// TIA Portal V20 program export: 0 tag tables, 0 data types, 5 data blocks, 15 code blocks (in call order from the OBs), 9 instance data blocks

DATA_BLOCK "Data_State2"   // DB12
{ S7_Optimized_Access := 'FALSE' }
   VAR
      state1 : "UDT_Flowmeter_Status";
      state_2 : "UDT_Flowmeter_Stoe";
   END_VAR
BEGIN
END_DATA_BLOCK

DATA_BLOCK "Date and Time"   // DB3
{ S7_Optimized_Access := 'FALSE' }
AUTHOR : L.P.
// stored: AutoNumber false
   VAR RETAIN
      MEM : Struct
         "set by host" : Bool;
         "HM imp set by host" : Bool;
         "HM imp set by HMI" : Bool := false;
         "4" : Bool := false;
         "5" : Bool := false;
         "6" : Bool := false;
         "7" : Bool := false;
         "8" : Bool := false;
         "9" : Bool := false;
         "10" : Bool := false;
      END_STRUCT;
      "STEP" : Struct
         "0" : Bool;
         "1" : Bool;
         "2" : Bool;
         "3" : Bool;
         "4" : Bool;
         "5" : Bool;
         "6" : Bool;
         "7" : Bool;
         "8" : Bool;
         "9" : Bool;
         "10" : Bool;
      END_STRUCT;
      T : Struct
         "1" { S7_SetPoint := 'True'} : IEC_TIMER;
         "2" { S7_SetPoint := 'True'} : IEC_TIMER;
         "3" { S7_SetPoint := 'True'} : IEC_TIMER;
         "4" { S7_SetPoint := 'True'} : IEC_TIMER;
         "5" { S7_SetPoint := 'True'} : IEC_TIMER;
         "6" { S7_SetPoint := 'True'} : IEC_TIMER;
         "7" { S7_SetPoint := 'True'} : IEC_TIMER;
         "8" { S7_SetPoint := 'True'} : IEC_TIMER;
         "9" { S7_SetPoint := 'True'} : IEC_TIMER;
         "10" { S7_SetPoint := 'True'} : IEC_TIMER;
      END_STRUCT;
      C : Struct
         "1" { S7_SetPoint := 'True'} : IEC_COUNTER;
         "2" { S7_SetPoint := 'True'} : IEC_COUNTER;
         "3" { S7_SetPoint := 'True'} : IEC_COUNTER;
         "4" { S7_SetPoint := 'True'} : IEC_COUNTER;
         "5" { S7_SetPoint := 'True'} : IEC_COUNTER;
         "6" { S7_SetPoint := 'True'} : IEC_COUNTER;
         "7" { S7_SetPoint := 'True'} : IEC_COUNTER;
         "8" { S7_SetPoint := 'True'} : IEC_COUNTER;
         "9" { S7_SetPoint := 'True'} : IEC_COUNTER;
         "10" { S7_SetPoint := 'True'} : IEC_COUNTER;
      END_STRUCT;
      DATA : Struct
         "in date OP" : Date;
         "in time OP" : Time_Of_Day;
         "in date and time" : DTL;
         "out date and time" : DTL;
         year : UInt;
         month : USInt;
         day : USInt;
         hour : USInt;
         minute : USInt;
         second : USInt;
         millisecond : UInt;
         "day of week" : USInt;
         "day of year" : Int;
         "is Time Master" : Bool := true;
      END_STRUCT;
      BUTTON : Struct
         "set date and time" : Bool;
         "2" : Bool;
         "3" : Bool;
         "4" : Bool;
         "5" : Bool;
         "6" : Bool;
         "7" : Bool;
         "8" : Bool;
         "9" : Bool;
         "10" : Bool;
         "11" : Bool := false;
         "12" : Bool := false;
         "13" : Bool := false;
         "14" : Bool := false;
         "15" : Bool := false;
         "16" : Bool := false;
         "17" : Bool := false;
         "18" : Bool := false;
         "19" : Bool := false;
         "20" : Bool := false;
         "21" : Bool := false;
         "22" : Bool := false;
         "23" : Bool := false;
         "24" : Bool := false;
         "25" : Bool := false;
         "26" : Bool := false;
         "27" : Bool := false;
         "28" : Bool := false;
         "29" : Bool := false;
         "30" : Bool := false;
         "31" : Bool := false;
         "32" : Bool := false;
         "33" : Bool := false;
         "34" : Bool := false;
         "35" : Bool := false;
         "36" : Bool := false;
         "37" : Bool := false;
         "38" : Bool := false;
         "39" : Bool := false;
         "40" : Bool := false;
      END_STRUCT;
   END_VAR
BEGIN
END_DATA_BLOCK

DATA_BLOCK "GD_Data"   // DB11
{ S7_Optimized_Access := 'FALSE' }
   VAR RETAIN
      iocontrols : "UDT_Flowmeter_Steuern";
      CurrentValue { S7_SetPoint := 'True'} : DInt;
      zeit_ : Time;
      cycle_1s : Bool;
      count : Int;
      zeit : "UDT_RunTime_Status";
      settime { S7_SetPoint := 'True'} : "UDT_RunTime_Steuern";
      _Sec { S7_SetPoint := 'True'} : Int;
      _Min : Int;
      _Hours : Real;
      first_scan : Bool;
      startup_OK : Bool;
      Reset_Counter : Int;
      Date_Time_is_Lost : Bool;
      Counter_00 : DInt;
      Counter_01 : DInt;
      Testflowsensor_Status : "UDT_Flowmeter_Status";
      Testflowsensor_Control { S7_SetPoint := 'True'} : "UDT_Flowmeter_Steuern";
      Testfuelsensor_Stoe { S7_SetPoint := 'True'} : "UDT_Flowmeter_Stoe";
   END_VAR
BEGIN
END_DATA_BLOCK

DATA_BLOCK "General"   // DB2
{ S7_Optimized_Access := 'FALSE' }
AUTHOR : L.P.
// stored: AutoNumber false
   VAR RETAIN
      MEM : Struct
         off : Bool;
         on : Bool := false;
         "imp 50 ms" : Bool := false;
         "imp 100 ms" : Bool := false;
         "imp 200 ms" : Bool := false;
         "imp 400 ms" : Bool := false;
         "imp 500 ms" : Bool := false;
         "imp 800 ms" : Bool := false;
         "imp 1 s" : Bool := false;
         "imp 1,6 s" : Bool := false;
         "imp 2 s" : Bool := false;
         "HM imp 50 ms 1" : Bool := false;
         "HM imp 50 ms 2" : Bool := false;
         "HM imp 100 ms" : Bool := false;
         "HM imp 200 ms" : Bool := false;
         "HM imp 400 ms" : Bool := false;
         "HM imp 500 ms" : Bool := false;
         "HM imp 800 ms" : Bool := false;
         "HM imp 1 s" : Bool := false;
         "HM imp 1,6 s" : Bool := false;
         "HM imp 2 s" : Bool := false;
         "single pal" : Bool := false;
         "douple pal" : Bool := false;
         "warm start" : Bool := false;
         commissioning : Bool := false;
         "pal is model M5" : Bool;
         "pal is model M6" : Bool := false;
         "pal is model M7" : Bool := false;
         "29" : Bool := false;
         "pal is model M9" : Bool := false;
         "31" : Bool := false;
         "32" : Bool := false;
         "33" : Bool := false;
         "34" : Bool := false;
         "35" : Bool := false;
         "pal with stacker" : Bool := false;
         "37" : Bool := false;
         "38" : Bool := false;
         "39" : Bool := false;
         "pal with single infeed" : Bool := false;
         "pal with double infeed" : Bool := false;
         "42" : Bool := false;
         "43" : Bool := false;
         "stop cycle with button" : Bool := false;
         "drive RLP in safe position in stop cycle" : Bool := false;
         "46" : Bool := false;
         "47" : Bool := false;
         "48" : Bool := false;
         "49" : Bool := false;
         "wrapper with film clamp above" : Bool := false;
         "wrapper with film clamp on carriage" : Bool := false;
         "52" : Bool := false;
         "53" : Bool := false;
         "54" : Bool := false;
         "55" : Bool := false;
         "56" : Bool := false;
         "57" : Bool := false;
         "58" : Bool := false;
         "59" : Bool := false;
         "60" : Bool := false;
         "61" : Bool := false;
         "62" : Bool := false;
         "63" : Bool := false;
         "64" : Bool := false;
         "65" : Bool := false;
         "66" : Bool := false;
         "67" : Bool := false;
         "68" : Bool := false;
         "69" : Bool := false;
         "70" : Bool := false;
         "71" : Bool := false;
         "72" : Bool := false;
         "73" : Bool := false;
         "74" : Bool := false;
         "75" : Bool := false;
         "76" : Bool := false;
         "77" : Bool := false;
         "78" : Bool := false;
         "79" : Bool := false;
         "80" : Bool := false;
         "81" : Bool := false;
         "82" : Bool := false;
         "83" : Bool := false;
         "84" : Bool := false;
         "85" : Bool := false;
         "86" : Bool := false;
         "87" : Bool := false;
         "88" : Bool := false;
         "89" : Bool := false;
         "90" : Bool := false;
         "91" : Bool := false;
         "92" : Bool := false;
         "93" : Bool := false;
         "94" : Bool := false;
         "95" : Bool := false;
         "96" : Bool := false;
         "97" : Bool := false;
         "98" : Bool := false;
         "99" : Bool := false;
         "100" : Bool := false;
      END_STRUCT;
      "STEP" : Struct
         "0" : Bool;
         "1" : Bool;
         "2" : Bool := false;
         "3" : Bool := false;
         "4" : Bool := false;
         "5" : Bool := false;
         "6" : Bool := false;
         "7" : Bool := false;
         "8" : Bool := false;
         "9" : Bool := false;
         "10" : Bool := false;
      END_STRUCT;
      T : Struct
         "delay wachdog to FEE" { S7_SetPoint := 'True'} : IEC_TIMER;
         "delay no conection to FEE" { S7_SetPoint := 'True'} : IEC_TIMER;
         "3" { S7_SetPoint := 'True'} : IEC_TIMER;
         "4" { S7_SetPoint := 'True'} : IEC_TIMER;
         "5" { S7_SetPoint := 'True'} : IEC_TIMER;
         "6" { S7_SetPoint := 'True'} : IEC_TIMER;
         "7" { S7_SetPoint := 'True'} : IEC_TIMER;
         "8" { S7_SetPoint := 'True'} : IEC_TIMER;
         "9" { S7_SetPoint := 'True'} : IEC_TIMER;
         "10" { S7_SetPoint := 'True'} : IEC_TIMER;
         "11" { S7_SetPoint := 'True'} : IEC_TIMER;
         "12" { S7_SetPoint := 'True'} : IEC_TIMER;
         "13" { S7_SetPoint := 'True'} : IEC_TIMER;
         "14" { S7_SetPoint := 'True'} : IEC_TIMER;
         "15" { S7_SetPoint := 'True'} : IEC_TIMER;
         "16" { S7_SetPoint := 'True'} : IEC_TIMER;
         "17" { S7_SetPoint := 'True'} : IEC_TIMER;
         "18" { S7_SetPoint := 'True'} : IEC_TIMER;
         "19" { S7_SetPoint := 'True'} : IEC_TIMER;
         "20" { S7_SetPoint := 'True'} : IEC_TIMER;
         "21" { S7_SetPoint := 'True'} : IEC_TIMER;
         "22" { S7_SetPoint := 'True'} : IEC_TIMER;
         "23" { S7_SetPoint := 'True'} : IEC_TIMER;
         "24" { S7_SetPoint := 'True'} : IEC_TIMER;
         "25" { S7_SetPoint := 'True'} : IEC_TIMER;
         "26" { S7_SetPoint := 'True'} : IEC_TIMER;
         "27" { S7_SetPoint := 'True'} : IEC_TIMER;
         "28" { S7_SetPoint := 'True'} : IEC_TIMER;
         "29" { S7_SetPoint := 'True'} : IEC_TIMER;
         "30" { S7_SetPoint := 'True'} : IEC_TIMER;
      END_STRUCT;
      C : Struct
         "1" { S7_SetPoint := 'True'} : IEC_COUNTER;
         "2" { S7_SetPoint := 'True'} : IEC_COUNTER;
         "3" { S7_SetPoint := 'True'} : IEC_COUNTER;
         "4" { S7_SetPoint := 'True'} : IEC_COUNTER;
         "5" { S7_SetPoint := 'True'} : IEC_COUNTER;
         "6" { S7_SetPoint := 'True'} : IEC_COUNTER;
         "7" { S7_SetPoint := 'True'} : IEC_COUNTER;
         "8" { S7_SetPoint := 'True'} : IEC_COUNTER;
         "9" { S7_SetPoint := 'True'} : IEC_COUNTER;
         "10" { S7_SetPoint := 'True'} : IEC_COUNTER;
         "11" { S7_SetPoint := 'True'} : IEC_COUNTER;
         "12" { S7_SetPoint := 'True'} : IEC_COUNTER;
         "13" { S7_SetPoint := 'True'} : IEC_COUNTER;
         "14" { S7_SetPoint := 'True'} : IEC_COUNTER;
         "15" { S7_SetPoint := 'True'} : IEC_COUNTER;
         "16" { S7_SetPoint := 'True'} : IEC_COUNTER;
         "17" { S7_SetPoint := 'True'} : IEC_COUNTER;
         "18" { S7_SetPoint := 'True'} : IEC_COUNTER;
         "19" { S7_SetPoint := 'True'} : IEC_COUNTER;
         "20" { S7_SetPoint := 'True'} : IEC_COUNTER;
         "21" { S7_SetPoint := 'True'} : IEC_COUNTER;
         "22" { S7_SetPoint := 'True'} : IEC_COUNTER;
         "23" { S7_SetPoint := 'True'} : IEC_COUNTER;
         "24" { S7_SetPoint := 'True'} : IEC_COUNTER;
         "25" { S7_SetPoint := 'True'} : IEC_COUNTER;
         "26" { S7_SetPoint := 'True'} : IEC_COUNTER;
         "27" { S7_SetPoint := 'True'} : IEC_COUNTER;
         "28" { S7_SetPoint := 'True'} : IEC_COUNTER;
         "29" { S7_SetPoint := 'True'} : IEC_COUNTER;
         "30" { S7_SetPoint := 'True'} : IEC_COUNTER;
      END_STRUCT;
      DATA : Struct
         Byte1 : Byte;
         Byte2 : Byte := 16#0;
         Byte3 : Byte := 16#0;
         Byte4 : Byte := 16#0;
         Byte5 : Byte := 16#0;
         Byte6 : Byte := 16#0;
         Byte7 : Byte := 16#0;
         Byte8 : Byte := 16#0;
         Byte9 : Byte := 16#0;
         Byte10 : Byte := 16#0;
         "PAL NR" : Int;
         "Buffer Watchdog FEE" : Int;
         Int3 : Int := 0;
         Int4 : Int := 0;
         Int5 : Int := 0;
         Int6 : Int := 0;
         Int7 : Int;
         Int8 : Int := 0;
         Int9 : Int;
         Int10 : Int := 0;
         Dint1 : DInt;
         Dint2 : DInt := 0;
         Dint3 : DInt;
         Dint4 : DInt := 0;
         Dint5 : DInt;
         Dint6 : DInt := 0;
         Dint7 : DInt := 0;
         Dint8 : DInt := 0;
         Dint9 : DInt := 0;
         Dint10 : DInt := 0;
         "screen number HMI" : Array[0..4] of Int;
      END_STRUCT;
   END_VAR
BEGIN
END_DATA_BLOCK

DATA_BLOCK "I_Data"   // DB15
{ S7_Optimized_Access := 'FALSE' }
   VAR
      Data_IN : Struct
         Data_I_1 : Int := 1;
         Data_I_2 : Int := 2;
         Data_I_3 : Int := 3;
         Data_I_4 : Int := 4;
         Data_I_5 : Int := 5;
         Data_I_6 : Int := 6;
         Data_I_7 : Int := 7;
         Data_I_8 : Int := 8;
      END_STRUCT;
   END_VAR
BEGIN
END_DATA_BLOCK

ORGANIZATION_BLOCK "Main_1"   // OB1, LAD, ProgramCycle
TITLE = "Main Program Sweep (Cycle)"
{ S7_Optimized_Access := 'TRUE' }
// stored: SetENOAutomatically false
BEGIN

REGION Network 1
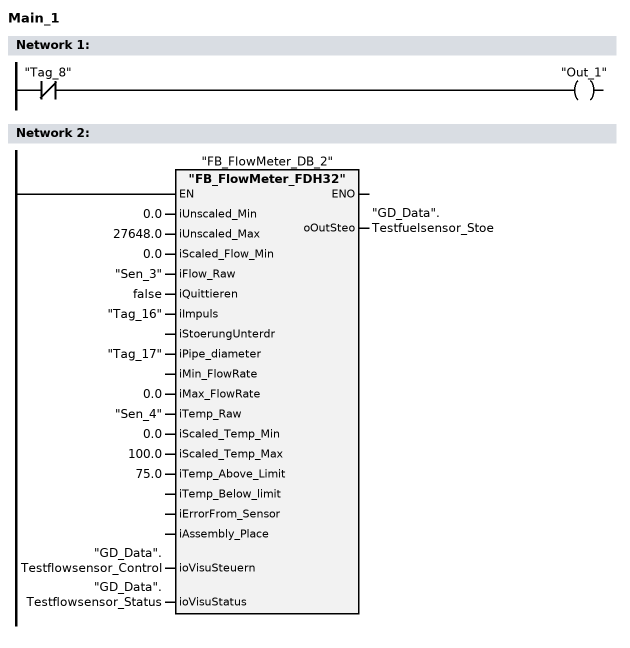
   RUNG wire#powerrail
      I_Contact( "Tag_8" )
      Coil( "Out_1" )
   END_RUNG
   // the same network as SCL:
   "Out_1" := NOT "Tag_8";
END_REGION

REGION Network 2
   RUNG wire#powerrail
      "FB_FlowMeter_DB_2"(iUnscaled_Min := 0.0, iUnscaled_Max := 27648.0, iScaled_Flow_Min := 0.0, iFlow_Raw := "Sen_3", iQuittieren := false, iImpuls := "Tag_16", iStoerungUnterdr :=, iPipe_diameter := "Tag_17", iMin_FlowRate :=, iMax_FlowRate := 0.0, iTemp_Raw := "Sen_4", iScaled_Temp_Min := 0.0, iScaled_Temp_Max := 100.0, iTemp_Above_Limit := 75.0, iTemp_Below_limit :=, iErrorFrom_Sensor :=, iAssembly_Place :=, ioVisuSteuern := "GD_Data".Testflowsensor_Control, ioVisuStatus := "GD_Data".Testflowsensor_Status, oOutSteo => "GD_Data".Testfuelsensor_Stoe)
   END_RUNG
   // the same network as SCL:
   "FB_FlowMeter_DB_2"(iUnscaled_Min := 0.0,   // "FB_FlowMeter_FDH32"
                       iUnscaled_Max := 27648.0,
                       iScaled_Flow_Min := 0.0,
                       iFlow_Raw := "Sen_3",
                       iQuittieren := false,
                       iImpuls := "Tag_16",
                       iPipe_diameter := "Tag_17",
                       iMax_FlowRate := 0.0,
                       iTemp_Raw := "Sen_4",
                       iScaled_Temp_Min := 0.0,
                       iScaled_Temp_Max := 100.0,
                       iTemp_Above_Limit := 75.0,
                       ioVisuSteuern := "GD_Data".Testflowsensor_Control,
                       ioVisuStatus := "GD_Data".Testflowsensor_Status,
                       oOutSteo => "GD_Data".Testfuelsensor_Stoe);
END_REGION
END_ORGANIZATION_BLOCK

FUNCTION_BLOCK "FB_FlowMeter_FDH32"   // FB10, LAD
{ S7_Optimized_Access := 'FALSE' }
// Durchfloss-Sensor FD-H Series 
// edited at 17.10.2025
// stored: SetENOAutomatically false
   VAR_INPUT
      iUnscaled_Min : Real;   // 0
      iUnscaled_Max : Real;   // 27648
      iScaled_Flow_Min : Real;
      iFlow_Raw : Int;
      iQuittieren : Bool;   // reset Fehler
      iImpuls : Bool;
      iStoerungUnterdr : Bool;
      iPipe_diameter : Bool;
      iMin_FlowRate : Real;
      iMax_FlowRate : Real;
      iTemp_Raw : Word;
      iScaled_Temp_Min : Real;
      iScaled_Temp_Max : Real;
      iTemp_Above_Limit { ExternalAccessible := 'False'; ExternalVisible := 'False'; ExternalWritable := 'False'} : Real;
      iTemp_Below_limit : Real;
      iErrorFrom_Sensor : Bool;   // Error signal from Sensor
      iAssembly_Place : String;
   END_VAR
   VAR_OUTPUT
      oOutSteo : "UDT_Flowmeter_Stoe";
   END_VAR
   VAR_IN_OUT
      ioVisuSteuern : "UDT_Flowmeter_Steuern";
      ioVisuStatus : "UDT_Flowmeter_Status";
   END_VAR
   VAR
      sFlow_ScaledValue : Real;
      sTemp_ScaledValue : Real;
      Buffer : Array[1..10] of Real;
      Index : DInt;
      Sum : Real;
      sScaled_Max : Real;
      i : Int;
      sAvg : Real;
      sCyclecount : Real;
      sOut_I : Int;
   END_VAR
   VAR_TEMP
      tVKE0 : Bool;
      tVKE1 : Bool;
      tbuffer01 : Int;
      tbuffer02 : Int;
      tbuffer03 : Int;
      tbuffer04 : DInt;
      tbuffer05 : Real;
      tbuffer06 : Word;
      tbuffer07 : Real;
      tNorm_FlowValue : Real;
      tNorm_TempValue : Real;
      tDrahtbruch1 : Bool;
      tDrahtbruch2 : Bool;
      tTempword : Word;
      tFlowword : Word;
      tSecond : Int;
      tMinute : Int;
      tHour : Int;
   END_VAR
   VAR_TEMP   // added for the SCL form of the ladder/FBD networks
      _w1 : Bool;
   END_VAR
BEGIN

REGION Network 1: Create tVKE1 Netzwek
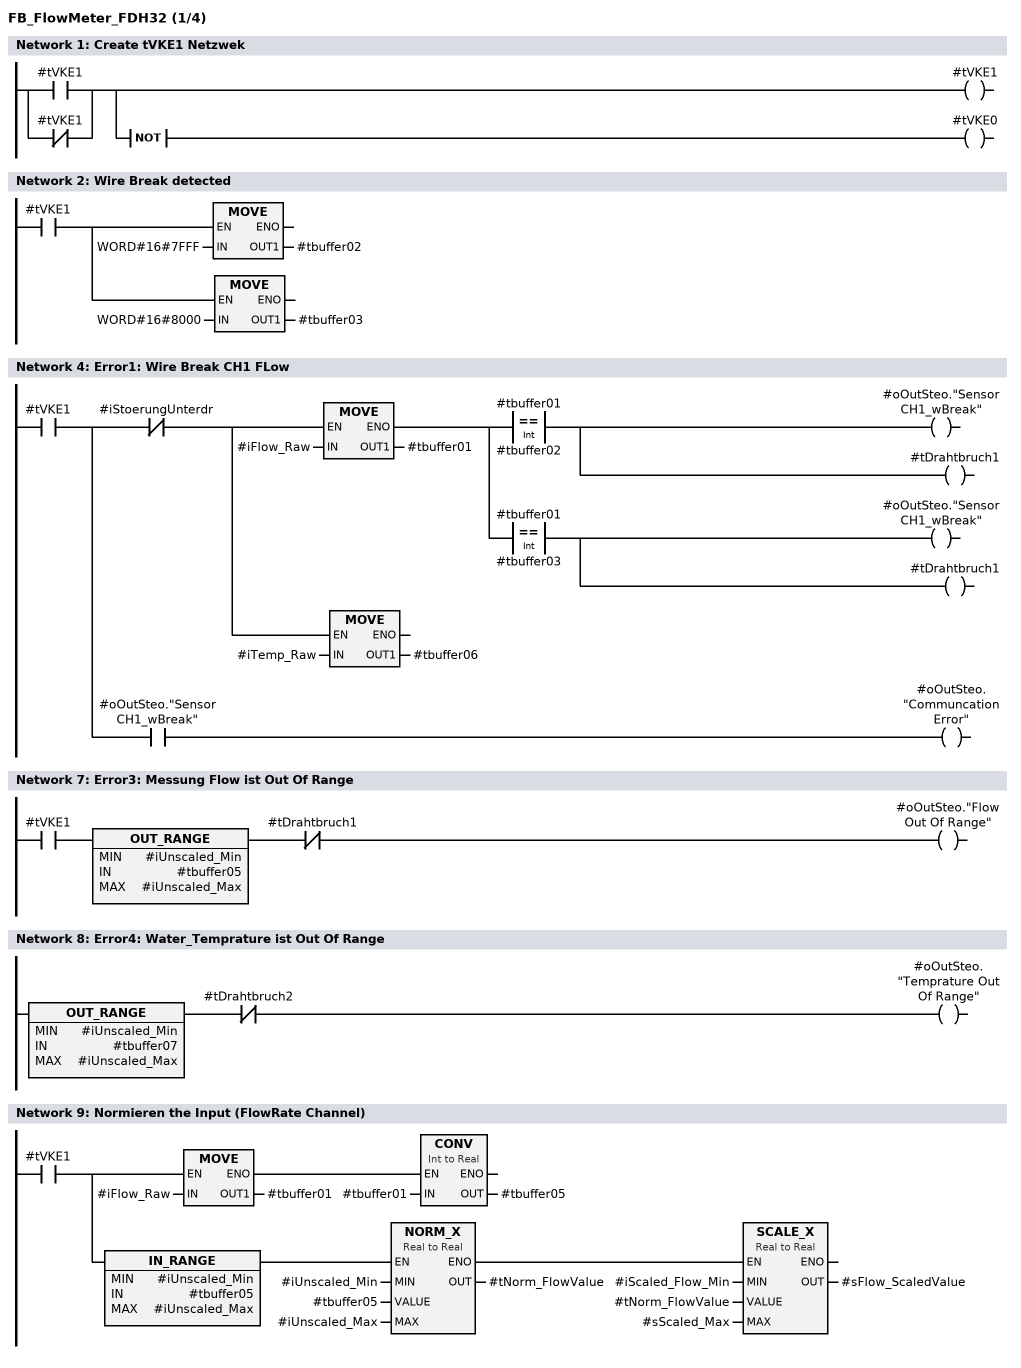
   RUNG wire#powerrail
      Contact( #tVKE1 )
      wire#w1
      Coil( #tVKE1 )
   END_RUNG
   RUNG wire#powerrail
      I_Contact( #tVKE1 )
   END_RUNG wire#w1
   RUNG wire#w1
      Not()
      Coil( #tVKE0 )
   END_RUNG
   // the same network as SCL:
   #tVKE1 := #tVKE1 OR NOT #tVKE1;
   #tVKE0 := NOT #tVKE1;
END_REGION

REGION Network 2: Wire Break detected
   RUNG wire#powerrail
      Contact( #tVKE1 )
      wire#w1
      { S7_GenerateENO := "TRUE" } Move(in := WORD#16#7FFF, out1 => #tbuffer02)
   END_RUNG
   RUNG wire#w1
      { S7_GenerateENO := "TRUE" } Move(in := WORD#16#8000, out1 => #tbuffer03)
   END_RUNG
   // the same network as SCL:
   IF #tVKE1 THEN
       #tbuffer02 := WORD#16#7FFF;
       #tbuffer03 := WORD#16#8000;
   END_IF;
END_REGION

REGION Network 3 (SCL): Reset All Error


   IF #iQuittieren THEN


       #oOutSteo."No Flow Detected"        := 0;
       #oOutSteo."Flow Rate Too Low"       := 0;
       #oOutSteo."Flow Rate Too Hight"     := 0;
       #oOutSteo."Sensor CH1_wBreak"       := 0;
       #oOutSteo."Sensor CH2_wBreak"       := 0;
       #oOutSteo."Temprature Above Limit"  := 0;
       #oOutSteo."Flow Out Of Range"       := 0;
       #oOutSteo."Calibration Error"       := 0;
       #oOutSteo."Air Bubles Detected"     := 0;
       #oOutSteo."Temprature Out Of Range" := 0;
       #oOutSteo."Temprature Below Limit"  := 0;
       #oOutSteo."Reverse Flow Detected"   := 0;
       #oOutSteo."Communcation Error"      := 0;
       #oOutSteo."Clogging or Blockage"    := 0;
       #oOutSteo."Sensor Overheating"      := 0;
       #oOutSteo."Dirty Sensor"            := 0;

   END_IF;
END_REGION

REGION Network 4: Error1: Wire Break CH1 FLow
   RUNG wire#powerrail
      Contact( #tVKE1 )
      wire#w1
      I_Contact( #iStoerungUnterdr )
      wire#w2
      { S7_GenerateENO := "TRUE" } Move(in := #iFlow_Raw, out1 => #tbuffer01)
      wire#w3
      { S7_Templates := "SrcType := Int" } EQ_Contact(in1 := #tbuffer01, in2 := #tbuffer02)
      wire#w4
      Coil( #oOutSteo."Sensor CH1_wBreak" )
   END_RUNG
   RUNG wire#w4
      Coil( #tDrahtbruch1 )
   END_RUNG
   RUNG wire#w3
      { S7_Templates := "SrcType := Int" } EQ_Contact(in1 := #tbuffer01, in2 := #tbuffer03)
      wire#w5
      Coil( #oOutSteo."Sensor CH1_wBreak" )
   END_RUNG
   RUNG wire#w5
      Coil( #tDrahtbruch1 )
   END_RUNG
   RUNG wire#w2
      { S7_GenerateENO := "TRUE" } Move(in := #iTemp_Raw, out1 => #tbuffer06)
   END_RUNG
   RUNG wire#w1
      Contact( #oOutSteo."Sensor CH1_wBreak" )
      Coil( #oOutSteo."Communcation Error" )
   END_RUNG
   // the same network as SCL:
   // ENO of a box is taken as its EN; it also drops when the box reports an error
   #_w1 := #tVKE1 AND NOT #iStoerungUnterdr;
   IF #_w1 THEN #tbuffer01 := #iFlow_Raw; END_IF;
   #oOutSteo."Sensor CH1_wBreak" := #_w1 AND (#tbuffer01 = #tbuffer02);
   #tDrahtbruch1 := #oOutSteo."Sensor CH1_wBreak";
   #oOutSteo."Sensor CH1_wBreak" := #_w1 AND (#tbuffer01 = #tbuffer03);
   #tDrahtbruch1 := #oOutSteo."Sensor CH1_wBreak";
   IF #_w1 THEN #tbuffer06 := #iTemp_Raw; END_IF;
   #oOutSteo."Communcation Error" := #tVKE1 AND #oOutSteo."Sensor CH1_wBreak";
END_REGION

REGION Network 5 (SCL): Evaluate Wire Break CH1 , CH2

   IF #iImpuls AND (#tDrahtbruch1 OR #tDrahtbruch2) THEN
       #tSecond := #tSecond + 1;

       IF #tSecond >= 60 THEN
           #tMinute := #tMinute + 1;
           #tSecond := 0;
       END_IF;

   END_IF;
END_REGION

REGION Network 6 (SCL): Error2: Wire Break CH2 Temprature
   IF #tbuffer06 = #tbuffer02 OR #tbuffer06 = #tbuffer03 THEN
       #tDrahtbruch2 := 1;
       #oOutSteo."Sensor CH2_wBreak" := 1;
   END_IF;
END_REGION

REGION Network 7: Error3: Messung Flow ist Out Of Range
   #oOutSteo."Flow Out Of Range" := #tVKE1 AND ((#tbuffer05 < #iUnscaled_Min) OR (#tbuffer05 > #iUnscaled_Max)) AND NOT #tDrahtbruch1;
END_REGION

REGION Network 8: Error4: Water_Temprature ist Out Of Range
   #oOutSteo."Temprature Out Of Range" := ((#tbuffer07 < #iUnscaled_Min) OR (#tbuffer07 > #iUnscaled_Max)) AND NOT #tDrahtbruch2;
END_REGION

REGION Network 9: Normieren the Input (FlowRate Channel)
   RUNG wire#powerrail
      Contact( #tVKE1 )
      wire#w1
      { S7_GenerateENO := "TRUE" } Move(in := #iFlow_Raw, out1 => #tbuffer01)
      { S7_Templates := "[SrcType := Int, DestType := Real]"; S7_GenerateENO := "TRUE" } Convert(in := #tbuffer01, out => #tbuffer05)
   END_RUNG
   RUNG wire#w1
      { S7_Templates := "SrcType := Real" } InRange(min := #iUnscaled_Min, in := #tbuffer05, max := #iUnscaled_Max)
      { S7_Templates := "[SrcType := Real, DestType := Real]"; S7_GenerateENO := "TRUE" } Normalize(min := #iUnscaled_Min, value := #tbuffer05, max := #iUnscaled_Max, out => #tNorm_FlowValue)
      { S7_Templates := "[SrcType := Real, DestType := Real]"; S7_GenerateENO := "TRUE" } Scale(min := #iScaled_Flow_Min, value := #tNorm_FlowValue, max := #sScaled_Max, out => #sFlow_ScaledValue)
   END_RUNG
   // the same network as SCL:
   // ENO of a box is taken as its EN; it also drops when the box reports an error
   IF #tVKE1 THEN
       #tbuffer01 := #iFlow_Raw;
       #tbuffer05 := INT_TO_REAL(#tbuffer01);
   END_IF;
   IF #tVKE1 AND (#iUnscaled_Min <= #tbuffer05) AND (#tbuffer05 <= #iUnscaled_Max) THEN
       #tNorm_FlowValue := NORM_X(MIN := #iUnscaled_Min, VALUE := #tbuffer05, MAX := #iUnscaled_Max);
       #sFlow_ScaledValue := SCALE_X(MIN := #iScaled_Flow_Min, VALUE := #tNorm_FlowValue, MAX := #sScaled_Max);
   END_IF;
END_REGION

REGION Network 10: Normieren & Scallieren the Water-Temprature
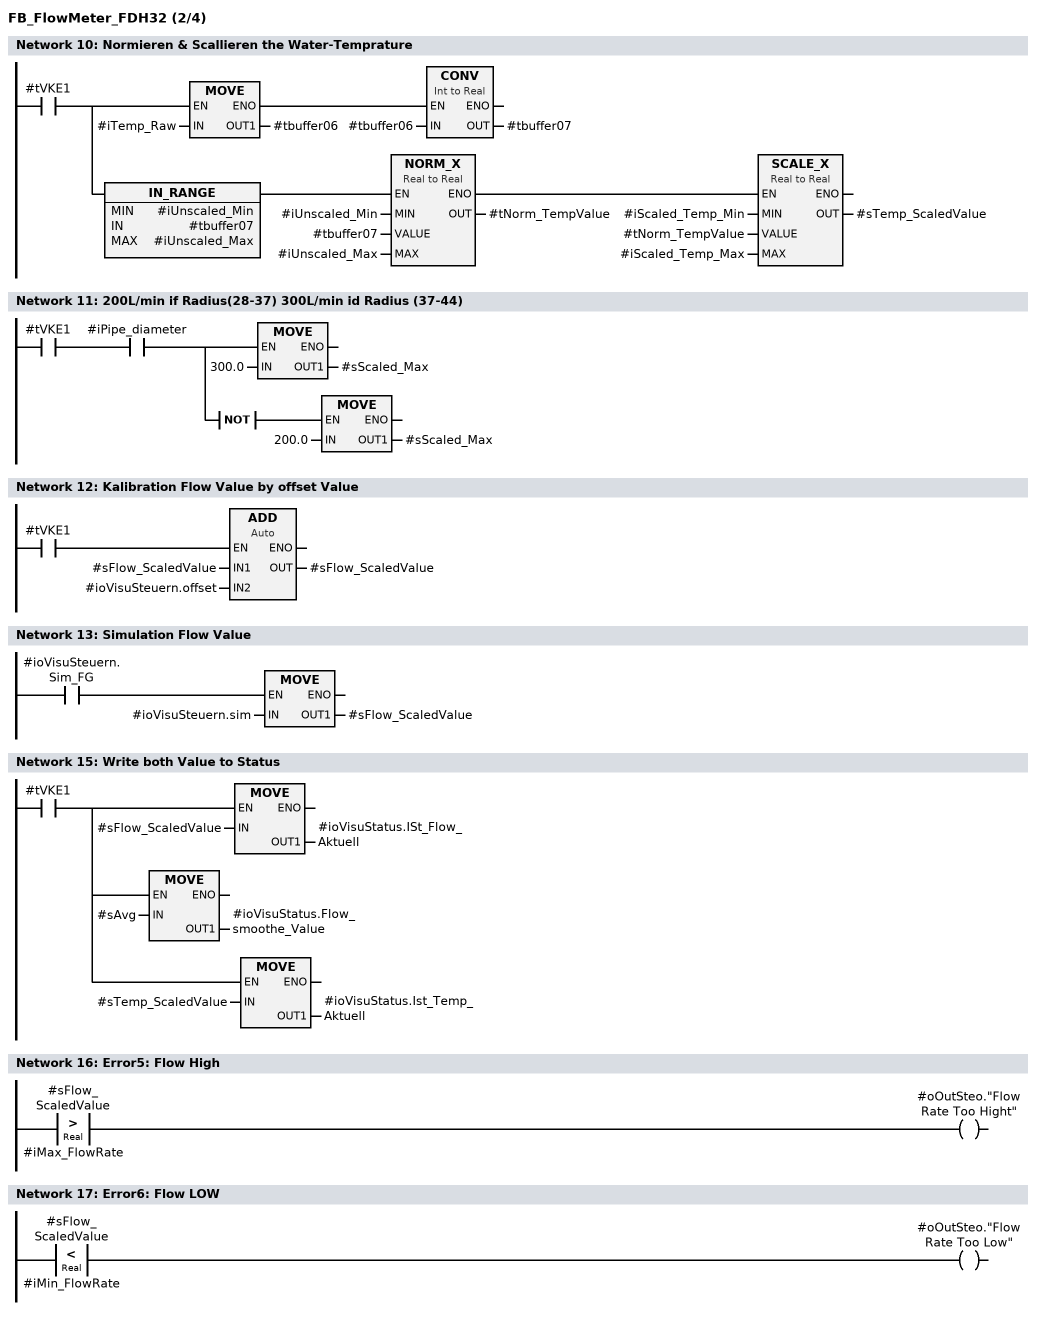
   RUNG wire#powerrail
      Contact( #tVKE1 )
      wire#w1
      { S7_GenerateENO := "TRUE" } Move(in := #iTemp_Raw, out1 => #tbuffer06)
      { S7_Templates := "[SrcType := Int, DestType := Real]"; S7_GenerateENO := "TRUE" } Convert(in := #tbuffer06, out => #tbuffer07)
   END_RUNG
   RUNG wire#w1
      { S7_Templates := "SrcType := Real" } InRange(min := #iUnscaled_Min, in := #tbuffer07, max := #iUnscaled_Max)
      { S7_Templates := "[SrcType := Real, DestType := Real]"; S7_GenerateENO := "TRUE" } Normalize(min := #iUnscaled_Min, value := #tbuffer07, max := #iUnscaled_Max, out => #tNorm_TempValue)
      { S7_Templates := "[SrcType := Real, DestType := Real]"; S7_GenerateENO := "TRUE" } Scale(min := #iScaled_Temp_Min, value := #tNorm_TempValue, max := #iScaled_Temp_Max, out => #sTemp_ScaledValue)
   END_RUNG
   // the same network as SCL:
   // ENO of a box is taken as its EN; it also drops when the box reports an error
   IF #tVKE1 THEN
       #tbuffer06 := #iTemp_Raw;
       #tbuffer07 := INT_TO_REAL(#tbuffer06);
   END_IF;
   IF #tVKE1 AND (#iUnscaled_Min <= #tbuffer07) AND (#tbuffer07 <= #iUnscaled_Max) THEN
       #tNorm_TempValue := NORM_X(MIN := #iUnscaled_Min, VALUE := #tbuffer07, MAX := #iUnscaled_Max);
       #sTemp_ScaledValue := SCALE_X(MIN := #iScaled_Temp_Min, VALUE := #tNorm_TempValue, MAX := #iScaled_Temp_Max);
   END_IF;
END_REGION

REGION Network 11: 200L/min if Radius(28-37) 300L/min id Radius (37-44)
   RUNG wire#powerrail
      Contact( #tVKE1 )
      Contact( #iPipe_diameter )
      wire#w1
      { S7_GenerateENO := "TRUE" } Move(in := 300.0, out1 => #sScaled_Max)
   END_RUNG
   RUNG wire#w1
      Not()
      { S7_GenerateENO := "TRUE" } Move(in := 200.0, out1 => #sScaled_Max)
   END_RUNG
   // the same network as SCL:
   #_w1 := #tVKE1 AND #iPipe_diameter;
   IF #_w1 THEN #sScaled_Max := 300.0; END_IF;
   IF NOT #_w1 THEN #sScaled_Max := 200.0; END_IF;
END_REGION

REGION Network 12: Kalibration Flow Value by offset Value
   RUNG wire#powerrail
      Contact( #tVKE1 )
      { S7_GenerateENO := "TRUE" } Add(in1 := #sFlow_ScaledValue, in2 := #ioVisuSteuern.offset, out => #sFlow_ScaledValue)
   END_RUNG
   // the same network as SCL:
   IF #tVKE1 THEN #sFlow_ScaledValue := #sFlow_ScaledValue + #ioVisuSteuern.offset; END_IF;
END_REGION

REGION Network 13: Simulation Flow Value
   RUNG wire#powerrail
      Contact( #ioVisuSteuern.Sim_FG )
      { S7_GenerateENO := "TRUE" } Move(in := #ioVisuSteuern.sim, out1 => #sFlow_ScaledValue)
   END_RUNG
   // the same network as SCL:
   IF #ioVisuSteuern.Sim_FG THEN #sFlow_ScaledValue := #ioVisuSteuern.sim; END_IF;
END_REGION

REGION Network 14 (SCL): Smoothing the Outsignal
   #sCyclecount := #sCyclecount + 1;

   IF #sCyclecount = 1 THEN
       FOR #i := 1 TO 10 DO
           #Buffer[#i] := #sFlow_ScaledValue;
       END_FOR;

       #Sum := #sFlow_ScaledValue * 10.0;
       #Index := 1;
       #sAvg := #sFlow_ScaledValue;

   ELSE

       #Sum := #Sum - #Buffer[#Index];
       #Buffer[#Index] := #sFlow_ScaledValue;
       #Sum := #Sum + #sFlow_ScaledValue;
       #sAvg := #Sum / 10.0;

       #Index := #Index + 1;
       IF #Index > 10 THEN
           #Index := 1;
       END_IF;
   END_IF;
END_REGION

REGION Network 15: Write both Value to Status
   RUNG wire#powerrail
      Contact( #tVKE1 )
      wire#w1
      { S7_GenerateENO := "TRUE" } Move(in := #sFlow_ScaledValue, out1 => #ioVisuStatus.ISt_Flow_Aktuell)
   END_RUNG
   RUNG wire#w1
      { S7_GenerateENO := "TRUE" } Move(in := #sAvg, out1 => #ioVisuStatus.Flow_smoothe_Value)
   END_RUNG
   RUNG wire#w1
      { S7_GenerateENO := "TRUE" } Move(in := #sTemp_ScaledValue, out1 => #ioVisuStatus.Ist_Temp_Aktuell)
   END_RUNG
   // the same network as SCL:
   IF #tVKE1 THEN
       #ioVisuStatus.ISt_Flow_Aktuell := #sFlow_ScaledValue;
       #ioVisuStatus.Flow_smoothe_Value := #sAvg;
       #ioVisuStatus.Ist_Temp_Aktuell := #sTemp_ScaledValue;
   END_IF;
END_REGION

REGION Network 16: Error5: Flow High
   RUNG wire#powerrail
      { S7_Templates := "SrcType := Real" } GT_Contact(in1 := #sFlow_ScaledValue, in2 := #iMax_FlowRate)
      Coil( #oOutSteo."Flow Rate Too Hight" )
   END_RUNG
   // the same network as SCL:
   #oOutSteo."Flow Rate Too Hight" := #sFlow_ScaledValue > #iMax_FlowRate;
END_REGION

REGION Network 17: Error6: Flow LOW
   RUNG wire#powerrail
      { S7_Templates := "SrcType := Real" } LT_Contact(in1 := #sFlow_ScaledValue, in2 := #iMin_FlowRate)
      Coil( #oOutSteo."Flow Rate Too Low" )
   END_RUNG
   // the same network as SCL:
   #oOutSteo."Flow Rate Too Low" := #sFlow_ScaledValue < #iMin_FlowRate;
END_REGION

REGION Network 18: Error7: Temp High
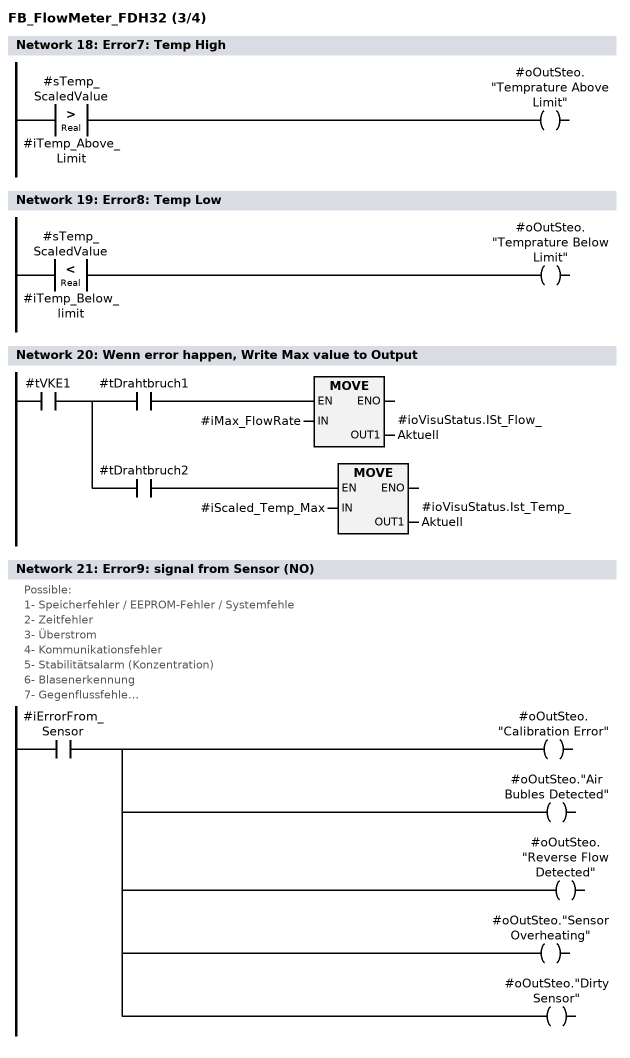
   RUNG wire#powerrail
      { S7_Templates := "SrcType := Real" } GT_Contact(in1 := #sTemp_ScaledValue, in2 := #iTemp_Above_Limit)
      Coil( #oOutSteo."Temprature Above Limit" )
   END_RUNG
   // the same network as SCL:
   #oOutSteo."Temprature Above Limit" := #sTemp_ScaledValue > #iTemp_Above_Limit;
END_REGION

REGION Network 19: Error8: Temp Low
   RUNG wire#powerrail
      { S7_Templates := "SrcType := Real" } LT_Contact(in1 := #sTemp_ScaledValue, in2 := #iTemp_Below_limit)
      Coil( #oOutSteo."Temprature Below Limit" )
   END_RUNG
   // the same network as SCL:
   #oOutSteo."Temprature Below Limit" := #sTemp_ScaledValue < #iTemp_Below_limit;
END_REGION

REGION Network 20: Wenn error happen, Write Max value to Output
   RUNG wire#powerrail
      Contact( #tVKE1 )
      wire#w1
      Contact( #tDrahtbruch1 )
      { S7_GenerateENO := "TRUE" } Move(in := #iMax_FlowRate, out1 => #ioVisuStatus.ISt_Flow_Aktuell)
   END_RUNG
   RUNG wire#w1
      Contact( #tDrahtbruch2 )
      { S7_GenerateENO := "TRUE" } Move(in := #iScaled_Temp_Max, out1 => #ioVisuStatus.Ist_Temp_Aktuell)
   END_RUNG
   // the same network as SCL:
   IF #tVKE1 AND #tDrahtbruch1 THEN #ioVisuStatus.ISt_Flow_Aktuell := #iMax_FlowRate; END_IF;
   IF #tVKE1 AND #tDrahtbruch2 THEN #ioVisuStatus.Ist_Temp_Aktuell := #iScaled_Temp_Max; END_IF;
END_REGION

REGION Network 21: Error9: signal from Sensor (NO)
   // Possible:
   // 1- Speicherfehler / EEPROM-Fehler / Systemfehle
   // 2- Zeitfehler 
   // 3- Überstrom
   // 4- Kommunikationsfehler
   // 5- Stabilitätsalarm (Konzentration)
   // 6- Blasenerkennung
   // 7- Gegenflussfehler
   // 8- Außerhalb des Erkennungsbereichs Temperatur
   RUNG wire#powerrail
      Contact( #iErrorFrom_Sensor )
      wire#w1
      Coil( #oOutSteo."Calibration Error" )
   END_RUNG
   RUNG wire#w1
      Coil( #oOutSteo."Air Bubles Detected" )
   END_RUNG
   RUNG wire#w1
      Coil( #oOutSteo."Reverse Flow Detected" )
   END_RUNG
   RUNG wire#w1
      Coil( #oOutSteo."Sensor Overheating" )
   END_RUNG
   RUNG wire#w1
      Coil( #oOutSteo."Dirty Sensor" )
   END_RUNG
   // the same network as SCL:
   #oOutSteo."Calibration Error" := #iErrorFrom_Sensor;
   #oOutSteo."Air Bubles Detected" := #iErrorFrom_Sensor;
   #oOutSteo."Reverse Flow Detected" := #iErrorFrom_Sensor;
   #oOutSteo."Sensor Overheating" := #iErrorFrom_Sensor;
   #oOutSteo."Dirty Sensor" := #iErrorFrom_Sensor;
END_REGION

REGION Network 22 (SCL): Error_Bit to word
   REGION _BitToWord

       #tFlowword := 0;

       IF #oOutSteo."No Flow Detected" THEN
           #tFlowword := #tFlowword OR W#16#1;
       END_IF;

       IF #oOutSteo."Flow Rate Too Low" THEN
           #tFlowword := #tFlowword OR W#16#2;
       END_IF;

       IF #oOutSteo."Flow Rate Too Hight" THEN
           #tFlowword := #tFlowword OR W#16#4;
       END_IF;

       IF #oOutSteo."Sensor CH1_wBreak" THEN
           #tFlowword := #tFlowword OR W#16#8;
       END_IF;

       IF #oOutSteo."Sensor CH2_wBreak" THEN
           #tFlowword := #tFlowword OR W#16#10;
       END_IF;

       IF #oOutSteo."Temprature Above Limit" THEN
           #tFlowword := #tFlowword OR W#16#20;
       END_IF;

       IF #oOutSteo."Flow Out Of Range" THEN
           #tFlowword := #tFlowword OR W#16#40;
       END_IF;

       IF #oOutSteo."Calibration Error" THEN
           #tFlowword := #tFlowword OR W#16#80;
       END_IF;

       IF #oOutSteo."Air Bubles Detected" THEN
           #tFlowword := #tFlowword OR W#16#100;
       END_IF;

       IF #oOutSteo."Temprature Out Of Range" THEN
           #tFlowword := #tFlowword OR W#16#200;
       END_IF;

       IF #oOutSteo."Temprature Below Limit" THEN
           #tFlowword := #tFlowword OR W#16#400;
       END_IF;

       IF #oOutSteo."Reverse Flow Detected" THEN
           #tFlowword := #tFlowword OR W#16#800;
       END_IF;

       IF #oOutSteo."Communcation Error" THEN
           #tFlowword := #tFlowword OR W#16#1000;
       END_IF;

       IF #oOutSteo."Clogging or Blockage" THEN
           #tFlowword := #tFlowword OR W#16#2000;
       END_IF;

       IF #oOutSteo."Sensor Overheating" THEN
           #tFlowword := #tFlowword OR W#16#4000;
       END_IF;

       IF #oOutSteo."Dirty Sensor" THEN
           #tFlowword := #tFlowword OR W#16#8000;
       END_IF;

       #sOut_I := WORD_TO_INT(#tFlowword);

   END_REGION
END_REGION

REGION Network 23 (SCL): Move Steo to Status

   #ioVisuStatus.MESS_DB_STOE := #tFlowword <> 0;
END_REGION

REGION Network 24 (SCL): Visu Farbe_NO Error

   // No Error  Green
   IF #tFlowword  = 0 THEN
       #ioVisuStatus.VISU_FARBE_Flow := 1;

   END_IF;
END_REGION

REGION Network 25: Visu Farbe_Warning
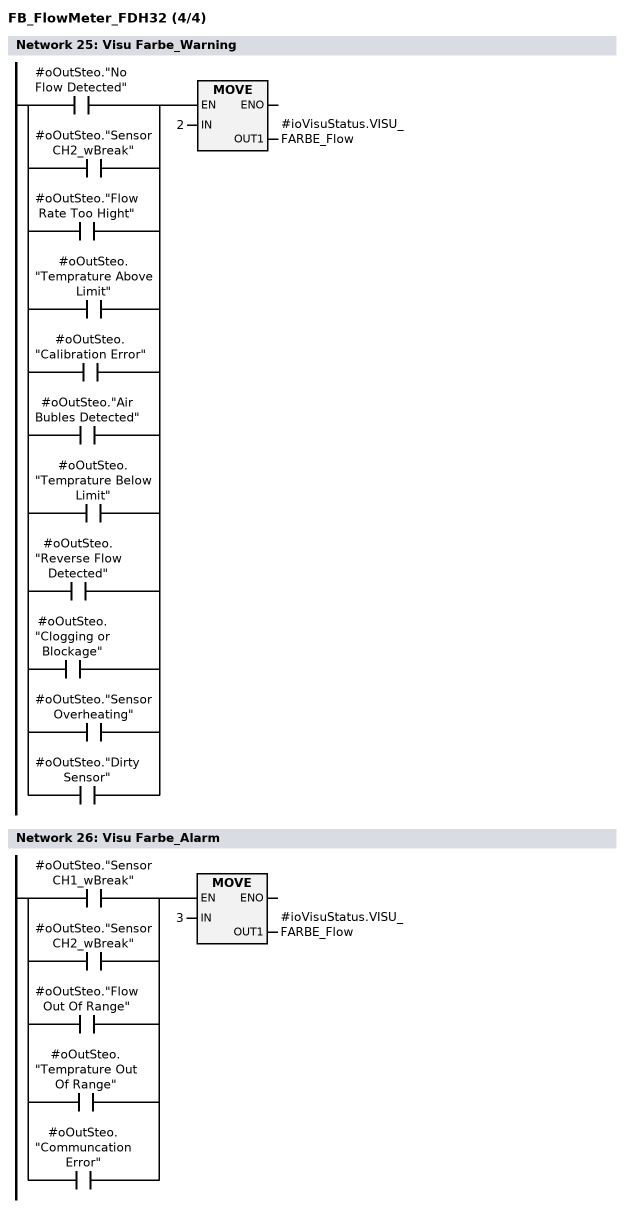
   RUNG wire#powerrail
      Contact( #oOutSteo."No Flow Detected" )
      wire#w1
      { S7_GenerateENO := "TRUE" } Move(in := 2, out1 => #ioVisuStatus.VISU_FARBE_Flow)
   END_RUNG
   RUNG wire#powerrail
      Contact( #oOutSteo."Sensor CH2_wBreak" )
   END_RUNG wire#w1
   RUNG wire#powerrail
      Contact( #oOutSteo."Flow Rate Too Hight" )
   END_RUNG wire#w1
   RUNG wire#powerrail
      Contact( #oOutSteo."Temprature Above Limit" )
   END_RUNG wire#w1
   RUNG wire#powerrail
      Contact( #oOutSteo."Calibration Error" )
   END_RUNG wire#w1
   RUNG wire#powerrail
      Contact( #oOutSteo."Air Bubles Detected" )
   END_RUNG wire#w1
   RUNG wire#powerrail
      Contact( #oOutSteo."Temprature Below Limit" )
   END_RUNG wire#w1
   RUNG wire#powerrail
      Contact( #oOutSteo."Reverse Flow Detected" )
   END_RUNG wire#w1
   RUNG wire#powerrail
      Contact( #oOutSteo."Clogging or Blockage" )
   END_RUNG wire#w1
   RUNG wire#powerrail
      Contact( #oOutSteo."Sensor Overheating" )
   END_RUNG wire#w1
   RUNG wire#powerrail
      Contact( #oOutSteo."Dirty Sensor" )
   END_RUNG wire#w1
   // the same network as SCL:
   IF #oOutSteo."No Flow Detected" OR #oOutSteo."Sensor CH2_wBreak" OR #oOutSteo."Flow Rate Too Hight" OR #oOutSteo."Temprature Above Limit" OR #oOutSteo."Calibration Error" OR #oOutSteo."Air Bubles Detected" OR #oOutSteo."Temprature Below Limit" OR #oOutSteo."Reverse Flow Detected" OR #oOutSteo."Clogging or Blockage" OR #oOutSteo."Sensor Overheating" OR #oOutSteo."Dirty Sensor" THEN
       #ioVisuStatus.VISU_FARBE_Flow := 2;
   END_IF;
END_REGION

REGION Network 26: Visu Farbe_Alarm
   RUNG wire#powerrail
      Contact( #oOutSteo."Sensor CH1_wBreak" )
      wire#w1
      { S7_GenerateENO := "TRUE" } Move(in := 3, out1 => #ioVisuStatus.VISU_FARBE_Flow)
   END_RUNG
   RUNG wire#powerrail
      Contact( #oOutSteo."Sensor CH2_wBreak" )
   END_RUNG wire#w1
   RUNG wire#powerrail
      Contact( #oOutSteo."Flow Out Of Range" )
   END_RUNG wire#w1
   RUNG wire#powerrail
      Contact( #oOutSteo."Temprature Out Of Range" )
   END_RUNG wire#w1
   RUNG wire#powerrail
      Contact( #oOutSteo."Communcation Error" )
   END_RUNG wire#w1
   // the same network as SCL:
   IF #oOutSteo."Sensor CH1_wBreak" OR #oOutSteo."Sensor CH2_wBreak" OR #oOutSteo."Flow Out Of Range" OR #oOutSteo."Temprature Out Of Range" OR #oOutSteo."Communcation Error" THEN
       #ioVisuStatus.VISU_FARBE_Flow := 3;
   END_IF;
END_REGION

REGION Network 27: End Baustein
END_REGION
END_FUNCTION_BLOCK

ORGANIZATION_BLOCK "CyclicInterrupt"   // OB35, LAD, CyclicInterrupt
{ S7_Optimized_Access := 'TRUE' }
// stored: AutoNumber false, SetENOAutomatically true
BEGIN
END_ORGANIZATION_BLOCK

ORGANIZATION_BLOCK "CyclicInterrupt_1"   // OB30, LAD, CyclicInterrupt
{ S7_Optimized_Access := 'TRUE' }
// stored: SetENOAutomatically false
BEGIN
END_ORGANIZATION_BLOCK

ORGANIZATION_BLOCK "DiagnosticErrorInterrupt_1"   // OB82, LAD, DiagnosticErrorInterrupt
{ S7_Optimized_Access := 'TRUE' }
// stored: SetENOAutomatically false
   VAR_INPUT
      IO_State : Word;   // IO state of the HW object
      LADDR : HW_ANY;   // Hardware identifier
      Channel : UInt;   // Channel number
      MultiError : Bool;   // =true if more than one error is present
   END_VAR
BEGIN
END_ORGANIZATION_BLOCK

ORGANIZATION_BLOCK "Startup_1"   // OB100, LAD, Startup
TITLE = "Complete Restart"
{ S7_Optimized_Access := 'TRUE' }
// stored: SetENOAutomatically false
   VAR_INPUT
      LostRetentive : Bool;   // True if retentive data are lost
      LostRTC : Bool;   // True if date and time are lost
   END_VAR
   VAR_TEMP
      NumberOf_Reset : Int;
   END_VAR
BEGIN

REGION Network 1
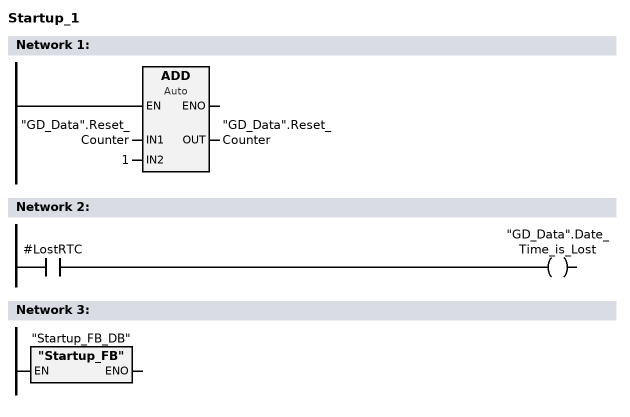
   RUNG wire#powerrail
      { S7_GenerateENO := "TRUE" } Add(in1 := "GD_Data".Reset_Counter, in2 := 1, out => "GD_Data".Reset_Counter)
   END_RUNG
   // the same network as SCL:
   "GD_Data".Reset_Counter := "GD_Data".Reset_Counter + 1;
END_REGION

REGION Network 2
   RUNG wire#powerrail
      Contact( #LostRTC )
      Coil( "GD_Data".Date_Time_is_Lost )
   END_RUNG
   // the same network as SCL:
   "GD_Data".Date_Time_is_Lost := #LostRTC;
END_REGION

REGION Network 3
   RUNG wire#powerrail
      "Startup_FB_DB"()
   END_RUNG
   // the same network as SCL:
   "Startup_FB_DB"();   // "Startup_FB"
END_REGION
END_ORGANIZATION_BLOCK

FUNCTION_BLOCK "Startup_FB"   // FB9, LAD
{ S7_Optimized_Access := 'TRUE' }
// stored: SetENOAutomatically false
BEGIN

REGION Network 1 (SCL)

   "R_TRIG_DB"(CLK:="FirstScan");
   IF "R_TRIG_DB".Q = 1 THEN
       "GD_Data".Counter_00 := "GD_Data".Counter_00 +1
       ;
   END_IF;
END_REGION
END_FUNCTION_BLOCK

ORGANIZATION_BLOCK "TimeErrorInterrupt_1"   // OB80, LAD, TimeErrorInterrupt
{ S7_Optimized_Access := 'TRUE' }
// stored: SetENOAutomatically false
   VAR_INPUT
      Fault_ID : Byte;   // Fault identifier
      Csg_OBnr : OB_ANY;   // Number of OB causing the error
      Csg_Prio : UInt;   // Priority of OB causing the error
   END_VAR
BEGIN
END_ORGANIZATION_BLOCK

FUNCTION_BLOCK "FB_Fuel_Stand"   // FB1, FBD
{ S7_Optimized_Access := 'TRUE' }
// stored: SetENOAutomatically false
   VAR_INPUT
      iUnscaledMin : Real;
      iUnscaledMax : Real;
      iScaledMin : Real;
      iOffset : Real;
      iUnscaledAktVal : Int;
      iQuittieren : Bool;
      iImpuls : Bool;
      iStoerungUnterdr : Bool;
      iPipe_diameter : Bool;
      iMaxFlowRate : Real;
      iTemp_Raw : Word;
      Temp_Min : Real;
      Temp_Max : Real;
      Refrence_Temp : Real;
      iAssembly_Place : String;
   END_VAR
   VAR_OUTPUT
      outputfehler : "UDT_Flowmeter_Stoe";
   END_VAR
   VAR
      sFlowScaledValue : Real;
      eingang_80_plc : Bool;
      Buffer : Array[1..10] of Real;
      Index : DInt;
      Sum : Real;
      sScaledMax : Real;
      i : Int;
      sAvg : Real;
      bitte_schalte_an : Bool;
      sCyclecount : Real;
      IEC_Timer_0_Instance { S7_SetPoint := 'True'} : TON_TIME;
   END_VAR
   VAR_TEMP
      tVKE0 : Bool;
      tVKE1 : Bool;
      tdurchflussrate : Real;
      tbuffer01 : Int;
      tbuffer02 : Int;
      tbuffer03 : Int;
      tbuffer04 : DInt;
      tbuffer05 : Real;
      tbuffer06 : Word;
      tbuffer07 : Real;
      tNorm_FlowValue : Real;
      tNorm_TempValue : Real;
      "sensor-is-active" : Bool;
      tDrahtbruch : Bool;
   END_VAR
BEGIN

REGION Network 1
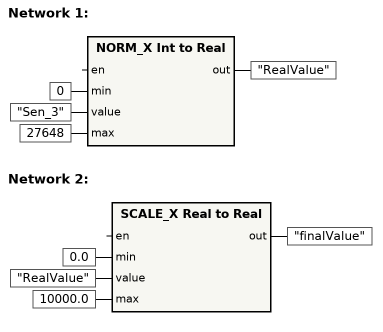
   "RealValue" := NORM_X(MIN := 0, VALUE := "Sen_3", MAX := 27648);
END_REGION

REGION Network 2
   "finalValue" := SCALE_X(MIN := 0.0, VALUE := "RealValue", MAX := 10000.0);
END_REGION
END_FUNCTION_BLOCK

FUNCTION_BLOCK "FB_Fuellstand"   // FB23, LAD
{ S7_Optimized_Access := 'FALSE' }
AUTHOR : F.EE
VERSION : 1.2
// stored: AutoNumber false, SetENOAutomatically false
   VAR_INPUT
      iScaledMin : Real;
      iScaledMax : Real;
      iUnscaledMin : Real;
      iUnscaledMax : Real;
      iOffset : Real;
      iUnscaledAktVal : Word;
      iStoerungUnterdr : Bool;
      iQuittieren : Bool;
      iImpuls : Bool;
   END_VAR
   VAR_OUTPUT
      tOutStoe : "UDT_FuellstandStoe";
   END_VAR
   VAR_IN_OUT
      ioVisuSteuern : "UDT_FuellstandSteuern";
      ioVisuStatus : "UDT_FuellstandStatus";
   END_VAR
   VAR
      sZeitDrahtbruch : Real;
      sAktPos : Real;
      sAktPosGlatt : Real;
      sDrahtbruch : Bool;
      sZeitEinsch : Real;
      sZeitAussch : Real;
      sEinschalt : Bool;
      sAusschalt : Bool;
      sStoerBit1 : Bool;
      SWertAlt : Real;
      sHmStoerBit1 : Bool;
      sImStoerBit1 : Bool;
   END_VAR
   VAR_TEMP
      tOffset : Real;
      tVKE1 : Bool;
      tVKE0 : Bool;
      tbuffer01 : Real;
      tbuffer02 : Real;
      tbuffer03 : Real;
      tbuffer04 : Real;
      tbuffer05 : Real;
      tbufferDI01 : DInt;
      tbufferI01 : Int;
      tbufferI02 : Int;
      tbufferI03 : Int;
      tSaveDI : DInt;
      tRetVal : Int;
      tDrahtbruch : Bool;
   END_VAR
   VAR_TEMP   // added for the SCL form of the ladder/FBD networks
      _w1 : Bool;
      _w2 : Bool;
   END_VAR
BEGIN

REGION Network 2
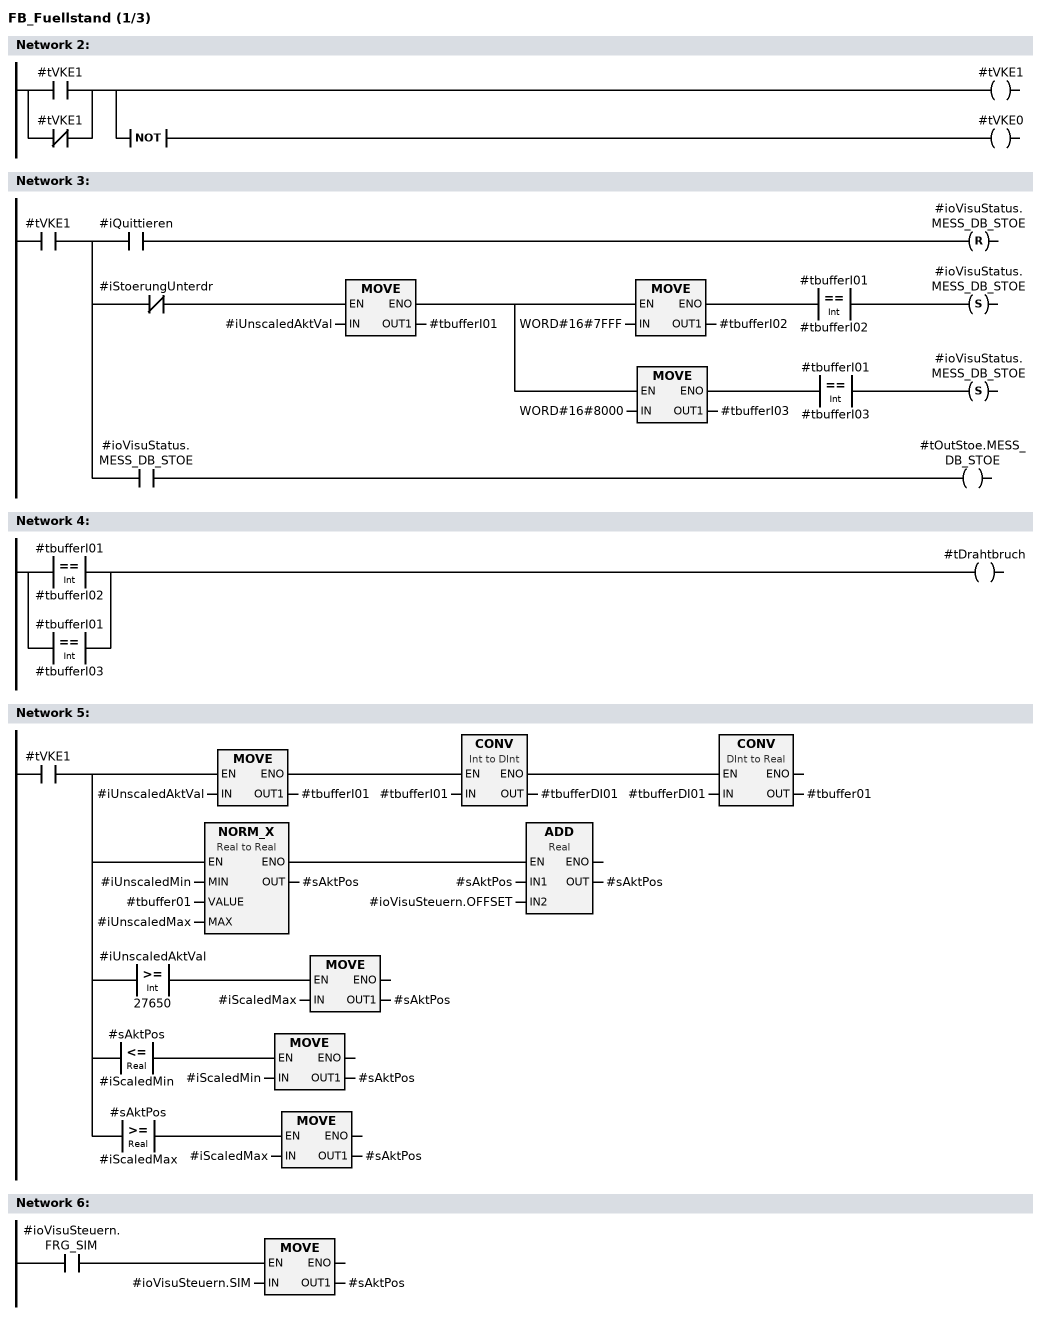
   RUNG wire#powerrail
      Contact( #tVKE1 )
      wire#w1
      Coil( #tVKE1 )
   END_RUNG
   RUNG wire#powerrail
      I_Contact( #tVKE1 )
   END_RUNG wire#w1
   RUNG wire#w1
      Not()
      Coil( #tVKE0 )
   END_RUNG
   // the same network as SCL:
   #tVKE1 := #tVKE1 OR NOT #tVKE1;
   #tVKE0 := NOT #tVKE1;
END_REGION

REGION Network 3
   RUNG wire#powerrail
      Contact( #tVKE1 )
      wire#w1
      Contact( #iQuittieren )
      R_Coil( #ioVisuStatus.MESS_DB_STOE )
   END_RUNG
   RUNG wire#w1
      I_Contact( #iStoerungUnterdr )
      { S7_GenerateENO := "TRUE" } Move(in := #iUnscaledAktVal, out1 => #tbufferI01)
      wire#w2
      { S7_GenerateENO := "TRUE" } Move(in := WORD#16#7FFF, out1 => #tbufferI02)
      { S7_Templates := "SrcType := Int" } EQ_Contact(in1 := #tbufferI01, in2 := #tbufferI02)
      S_Coil( #ioVisuStatus.MESS_DB_STOE )
   END_RUNG
   RUNG wire#w2
      { S7_GenerateENO := "TRUE" } Move(in := WORD#16#8000, out1 => #tbufferI03)
      { S7_Templates := "SrcType := Int" } EQ_Contact(in1 := #tbufferI01, in2 := #tbufferI03)
      S_Coil( #ioVisuStatus.MESS_DB_STOE )
   END_RUNG
   RUNG wire#w1
      Contact( #ioVisuStatus.MESS_DB_STOE )
      Coil( #tOutStoe.MESS_DB_STOE )
   END_RUNG
   // the same network as SCL:
   // ENO of a box is taken as its EN; it also drops when the box reports an error
   IF #tVKE1 AND #iQuittieren THEN #ioVisuStatus.MESS_DB_STOE := FALSE; END_IF;
   #_w1 := #tVKE1 AND NOT #iStoerungUnterdr;
   IF #_w1 THEN
       #tbufferI01 := #iUnscaledAktVal;
       #tbufferI02 := WORD#16#7FFF;
   END_IF;
   IF #_w1 AND (#tbufferI01 = #tbufferI02) THEN #ioVisuStatus.MESS_DB_STOE := TRUE; END_IF;
   IF #_w1 THEN #tbufferI03 := WORD#16#8000; END_IF;
   IF #_w1 AND (#tbufferI01 = #tbufferI03) THEN #ioVisuStatus.MESS_DB_STOE := TRUE; END_IF;
   #tOutStoe.MESS_DB_STOE := #tVKE1 AND #ioVisuStatus.MESS_DB_STOE;
END_REGION

REGION Network 4
   RUNG wire#powerrail
      { S7_Templates := "SrcType := Int" } EQ_Contact(in1 := #tbufferI01, in2 := #tbufferI02)
      wire#w1
      Coil( #tDrahtbruch )
   END_RUNG
   RUNG wire#powerrail
      { S7_Templates := "SrcType := Int" } EQ_Contact(in1 := #tbufferI01, in2 := #tbufferI03)
   END_RUNG wire#w1
   // the same network as SCL:
   #tDrahtbruch := (#tbufferI01 = #tbufferI02) OR (#tbufferI01 = #tbufferI03);
END_REGION

REGION Network 5
   RUNG wire#powerrail
      Contact( #tVKE1 )
      wire#w1
      { S7_GenerateENO := "TRUE" } Move(in := #iUnscaledAktVal, out1 => #tbufferI01)
      { S7_Templates := "[SrcType := Int, DestType := DInt]"; S7_GenerateENO := "TRUE" } Convert(in := #tbufferI01, out => #tbufferDI01)
      { S7_Templates := "[SrcType := DInt, DestType := Real]"; S7_GenerateENO := "TRUE" } Convert(in := #tbufferDI01, out => #tbuffer01)
   END_RUNG
   RUNG wire#w1
      { S7_Templates := "[SrcType := Real, DestType := Real]"; S7_GenerateENO := "TRUE" } Normalize(min := #iUnscaledMin, value := #tbuffer01, max := #iUnscaledMax, out => #sAktPos)
      { S7_Templates := "SrcType := Real"; S7_GenerateENO := "TRUE" } Add(in1 := #sAktPos, in2 := #ioVisuSteuern.OFFSET, out => #sAktPos)
   END_RUNG
   RUNG wire#w1
      { S7_Templates := "SrcType := Int" } GE_Contact(in1 := #iUnscaledAktVal, in2 := 27650)
      { S7_GenerateENO := "TRUE" } Move(in := #iScaledMax, out1 => #sAktPos)
   END_RUNG
   RUNG wire#w1
      { S7_Templates := "SrcType := Real" } LE_Contact(in1 := #sAktPos, in2 := #iScaledMin)
      { S7_GenerateENO := "TRUE" } Move(in := #iScaledMin, out1 => #sAktPos)
   END_RUNG
   RUNG wire#w1
      { S7_Templates := "SrcType := Real" } GE_Contact(in1 := #sAktPos, in2 := #iScaledMax)
      { S7_GenerateENO := "TRUE" } Move(in := #iScaledMax, out1 => #sAktPos)
   END_RUNG
   // the same network as SCL:
   // ENO of a box is taken as its EN; it also drops when the box reports an error
   IF #tVKE1 THEN
       #tbufferI01 := #iUnscaledAktVal;
       #tbufferDI01 := INT_TO_DINT(#tbufferI01);
       #tbuffer01 := DINT_TO_REAL(#tbufferDI01);
       #sAktPos := NORM_X(MIN := #iUnscaledMin, VALUE := #tbuffer01, MAX := #iUnscaledMax);
       #sAktPos := #sAktPos + #ioVisuSteuern.OFFSET;
   END_IF;
   IF #tVKE1 AND (#iUnscaledAktVal >= 27650) THEN #sAktPos := #iScaledMax; END_IF;
   IF #tVKE1 AND (#sAktPos <= #iScaledMin) THEN #sAktPos := #iScaledMin; END_IF;
   IF #tVKE1 AND (#sAktPos >= #iScaledMax) THEN #sAktPos := #iScaledMax; END_IF;
END_REGION

REGION Network 6
   RUNG wire#powerrail
      Contact( #ioVisuSteuern.FRG_SIM )
      { S7_GenerateENO := "TRUE" } Move(in := #ioVisuSteuern.SIM, out1 => #sAktPos)
   END_RUNG
   // the same network as SCL:
   IF #ioVisuSteuern.FRG_SIM THEN #sAktPos := #ioVisuSteuern.SIM; END_IF;
END_REGION

REGION Network 7
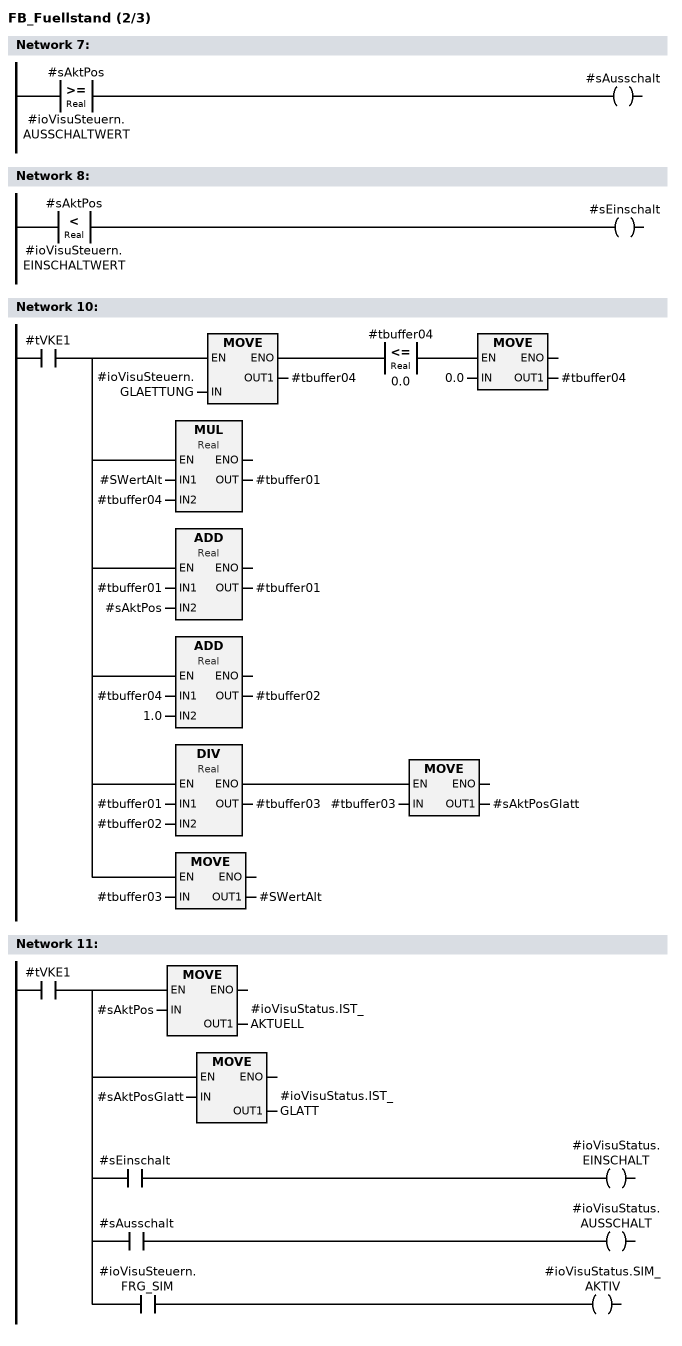
   RUNG wire#powerrail
      { S7_Templates := "SrcType := Real" } GE_Contact(in1 := #sAktPos, in2 := #ioVisuSteuern.AUSSCHALTWERT)
      Coil( #sAusschalt )
   END_RUNG
   // the same network as SCL:
   #sAusschalt := #sAktPos >= #ioVisuSteuern.AUSSCHALTWERT;
END_REGION

REGION Network 8
   RUNG wire#powerrail
      { S7_Templates := "SrcType := Real" } LT_Contact(in1 := #sAktPos, in2 := #ioVisuSteuern.EINSCHALTWERT)
      Coil( #sEinschalt )
   END_RUNG
   // the same network as SCL:
   #sEinschalt := #sAktPos < #ioVisuSteuern.EINSCHALTWERT;
END_REGION

REGION Network 9 (SCL)
   IF DINT_TO_DWORD(ROUND(#SWertAlt)) = 16#7FFFFFF THEN
       #SWertAlt := 0.0;
   END_IF;
END_REGION

REGION Network 10
   RUNG wire#powerrail
      Contact( #tVKE1 )
      wire#w1
      { S7_GenerateENO := "TRUE" } Move(in := #ioVisuSteuern.GLAETTUNG, out1 => #tbuffer04)
      { S7_Templates := "SrcType := Real" } LE_Contact(in1 := #tbuffer04, in2 := 0.0)
      { S7_GenerateENO := "TRUE" } Move(in := 0.0, out1 => #tbuffer04)
   END_RUNG
   RUNG wire#w1
      { S7_Templates := "SrcType := Real"; S7_GenerateENO := "TRUE" } Mul(in1 := #SWertAlt, in2 := #tbuffer04, out => #tbuffer01)
   END_RUNG
   RUNG wire#w1
      { S7_Templates := "SrcType := Real"; S7_GenerateENO := "TRUE" } Add(in1 := #tbuffer01, in2 := #sAktPos, out => #tbuffer01)
   END_RUNG
   RUNG wire#w1
      { S7_Templates := "SrcType := Real"; S7_GenerateENO := "TRUE" } Add(in1 := #tbuffer04, in2 := 1.0, out => #tbuffer02)
   END_RUNG
   RUNG wire#w1
      { S7_Templates := "SrcType := Real"; S7_GenerateENO := "TRUE" } Div(in1 := #tbuffer01, in2 := #tbuffer02, out => #tbuffer03)
      { S7_GenerateENO := "TRUE" } Move(in := #tbuffer03, out1 => #sAktPosGlatt)
   END_RUNG
   RUNG wire#w1
      { S7_GenerateENO := "TRUE" } Move(in := #tbuffer03, out1 => #SWertAlt)
   END_RUNG
   // the same network as SCL:
   // ENO of a box is taken as its EN; it also drops when the box reports an error
   IF #tVKE1 THEN #tbuffer04 := #ioVisuSteuern.GLAETTUNG; END_IF;
   IF #tVKE1 AND (#tbuffer04 <= 0.0) THEN #tbuffer04 := 0.0; END_IF;
   IF #tVKE1 THEN
       #tbuffer01 := #SWertAlt * #tbuffer04;
       #tbuffer01 := #tbuffer01 + #sAktPos;
       #tbuffer02 := #tbuffer04 + 1.0;
       #tbuffer03 := #tbuffer01 / #tbuffer02;
       #sAktPosGlatt := #tbuffer03;
       #SWertAlt := #tbuffer03;
   END_IF;
END_REGION

REGION Network 11
   RUNG wire#powerrail
      Contact( #tVKE1 )
      wire#w1
      { S7_GenerateENO := "TRUE" } Move(in := #sAktPos, out1 => #ioVisuStatus.IST_AKTUELL)
   END_RUNG
   RUNG wire#w1
      { S7_GenerateENO := "TRUE" } Move(in := #sAktPosGlatt, out1 => #ioVisuStatus.IST_GLATT)
   END_RUNG
   RUNG wire#w1
      Contact( #sEinschalt )
      Coil( #ioVisuStatus.EINSCHALT )
   END_RUNG
   RUNG wire#w1
      Contact( #sAusschalt )
      Coil( #ioVisuStatus.AUSSCHALT )
   END_RUNG
   RUNG wire#w1
      Contact( #ioVisuSteuern.FRG_SIM )
      Coil( #ioVisuStatus.SIM_AKTIV )
   END_RUNG
   // the same network as SCL:
   IF #tVKE1 THEN
       #ioVisuStatus.IST_AKTUELL := #sAktPos;
       #ioVisuStatus.IST_GLATT := #sAktPosGlatt;
   END_IF;
   #ioVisuStatus.EINSCHALT := #tVKE1 AND #sEinschalt;
   #ioVisuStatus.AUSSCHALT := #tVKE1 AND #sAusschalt;
   #ioVisuStatus.SIM_AKTIV := #tVKE1 AND #ioVisuSteuern.FRG_SIM;
END_REGION

REGION Network 12
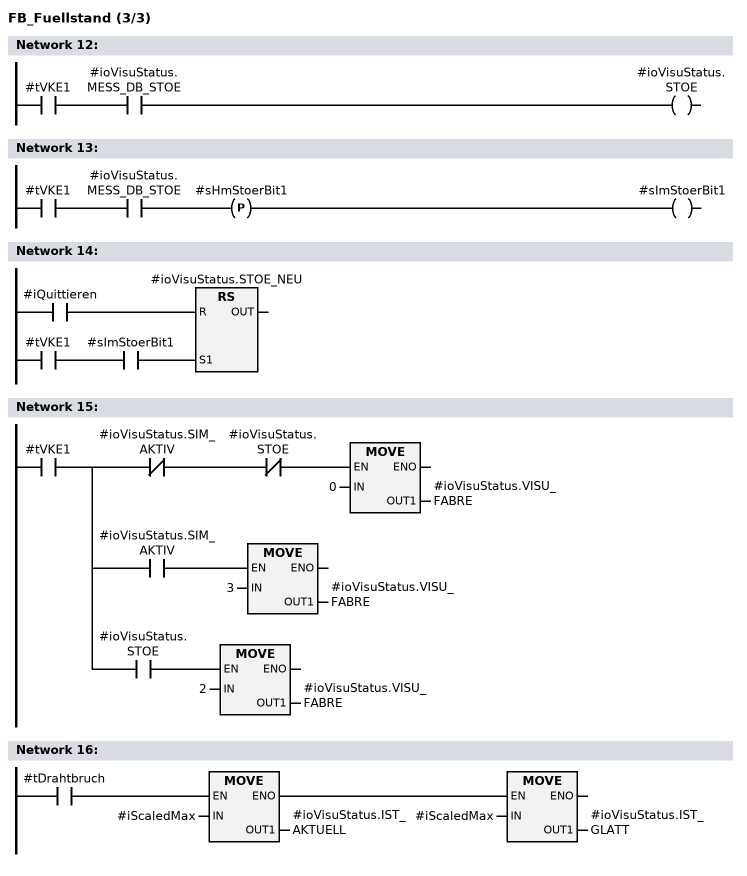
   RUNG wire#powerrail
      Contact( #tVKE1 )
      Contact( #ioVisuStatus.MESS_DB_STOE )
      Coil( #ioVisuStatus.STOE )
   END_RUNG
   // the same network as SCL:
   #ioVisuStatus.STOE := #tVKE1 AND #ioVisuStatus.MESS_DB_STOE;
END_REGION

REGION Network 13
   RUNG wire#powerrail
      Contact( #tVKE1 )
      Contact( #ioVisuStatus.MESS_DB_STOE )
      P_Trig( #sHmStoerBit1 )
      Coil( #sImStoerBit1 )
   END_RUNG
   // the same network as SCL:
   #_w1 := #tVKE1 AND #ioVisuStatus.MESS_DB_STOE;
   #_w2 := #_w1 AND NOT #sHmStoerBit1;   // rising edge
   #sHmStoerBit1 := #_w1;
   #sImStoerBit1 := #_w2;
END_REGION

REGION Network 14
   RUNG wire#powerrail
      Contact( #iQuittieren )
      S_RS(operand := #ioVisuStatus.STOE_NEU, s1 := wire#w1)
   END_RUNG
   RUNG wire#powerrail
      Contact( #tVKE1 )
      Contact( #sImStoerBit1 )
   END_RUNG wire#w1
   // the same network as SCL:
   IF #iQuittieren THEN
       #ioVisuStatus.STOE_NEU := FALSE;   // RS flip-flop
   END_IF;
   IF #tVKE1 AND #sImStoerBit1 THEN #ioVisuStatus.STOE_NEU := TRUE; END_IF;
END_REGION

REGION Network 15
   RUNG wire#powerrail
      Contact( #tVKE1 )
      wire#w1
      I_Contact( #ioVisuStatus.SIM_AKTIV )
      I_Contact( #ioVisuStatus.STOE )
      { S7_GenerateENO := "TRUE" } Move(in := 0, out1 => #ioVisuStatus.VISU_FABRE)
   END_RUNG
   RUNG wire#w1
      Contact( #ioVisuStatus.SIM_AKTIV )
      { S7_GenerateENO := "TRUE" } Move(in := 3, out1 => #ioVisuStatus.VISU_FABRE)
   END_RUNG
   RUNG wire#w1
      Contact( #ioVisuStatus.STOE )
      { S7_GenerateENO := "TRUE" } Move(in := 2, out1 => #ioVisuStatus.VISU_FABRE)
   END_RUNG
   // the same network as SCL:
   IF #tVKE1 AND NOT #ioVisuStatus.SIM_AKTIV AND NOT #ioVisuStatus.STOE THEN
       #ioVisuStatus.VISU_FABRE := 0;
   END_IF;
   IF #tVKE1 AND #ioVisuStatus.SIM_AKTIV THEN #ioVisuStatus.VISU_FABRE := 3; END_IF;
   IF #tVKE1 AND #ioVisuStatus.STOE THEN #ioVisuStatus.VISU_FABRE := 2; END_IF;
END_REGION

REGION Network 16
   RUNG wire#powerrail
      Contact( #tDrahtbruch )
      { S7_GenerateENO := "TRUE" } Move(in := #iScaledMax, out1 => #ioVisuStatus.IST_AKTUELL)
      { S7_GenerateENO := "TRUE" } Move(in := #iScaledMax, out1 => #ioVisuStatus.IST_GLATT)
   END_RUNG
   // the same network as SCL:
   // ENO of a box is taken as its EN; it also drops when the box reports an error
   IF #tDrahtbruch THEN
       #ioVisuStatus.IST_AKTUELL := #iScaledMax;
       #ioVisuStatus.IST_GLATT := #iScaledMax;
   END_IF;
END_REGION
END_FUNCTION_BLOCK

FUNCTION_BLOCK "Runtime"   // FB5, LAD
{ S7_Optimized_Access := 'TRUE' }
// stored: SetENOAutomatically false
   VAR_INPUT
      "iMotor Run Freedback" : Bool;
      iTakt_1Sec : Bool;
      iReset : Bool;
      iSetTime : Bool;
   END_VAR
   VAR_IN_OUT
      ioRun_Time_C : "UDT_RunTime_Steuern";
      ioRun_Time_S : "UDT_RunTime_Status";
      "ioReset_timer-Entern" : Bool;
   END_VAR
   VAR
      sMotoris_Enabled : Bool;
      P_TRIG : Bool;
   END_VAR
   VAR_TEMP
      tVKE1 : Bool;
      tVKE0 : Bool;
   END_VAR
   VAR CONSTANT
      cCounter_PV : Int := 60;
   END_VAR
   VAR_TEMP   // added for the SCL form of the ladder/FBD networks
      _w1 : Bool;
      _w2 : Bool;
   END_VAR
BEGIN

REGION Network 1: Create tVKE1 Netzwek
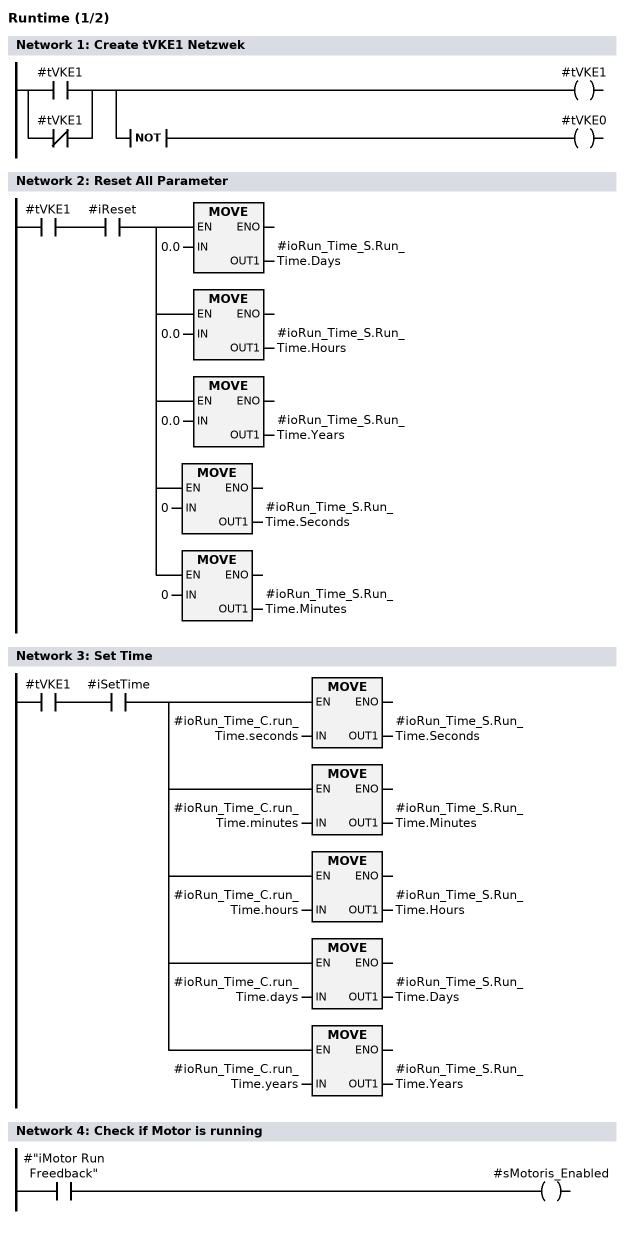
   RUNG wire#powerrail
      Contact( #tVKE1 )
      wire#w1
      Coil( #tVKE1 )
   END_RUNG
   RUNG wire#powerrail
      I_Contact( #tVKE1 )
   END_RUNG wire#w1
   RUNG wire#w1
      Not()
      Coil( #tVKE0 )
   END_RUNG
   // the same network as SCL:
   #tVKE1 := #tVKE1 OR NOT #tVKE1;
   #tVKE0 := NOT #tVKE1;
END_REGION

REGION Network 2: Reset All Parameter
   RUNG wire#powerrail
      Contact( #tVKE1 )
      Contact( #iReset )
      wire#w1
      { S7_GenerateENO := "TRUE" } Move(in := 0.0, out1 => #ioRun_Time_S.Run_Time.Days)
   END_RUNG
   RUNG wire#w1
      { S7_GenerateENO := "TRUE" } Move(in := 0.0, out1 => #ioRun_Time_S.Run_Time.Hours)
   END_RUNG
   RUNG wire#w1
      { S7_GenerateENO := "TRUE" } Move(in := 0.0, out1 => #ioRun_Time_S.Run_Time.Years)
   END_RUNG
   RUNG wire#w1
      { S7_GenerateENO := "TRUE" } Move(in := 0, out1 => #ioRun_Time_S.Run_Time.Seconds)
   END_RUNG
   RUNG wire#w1
      { S7_GenerateENO := "TRUE" } Move(in := 0, out1 => #ioRun_Time_S.Run_Time.Minutes)
   END_RUNG
   // the same network as SCL:
   IF #tVKE1 AND #iReset THEN
       #ioRun_Time_S.Run_Time.Days := 0.0;
       #ioRun_Time_S.Run_Time.Hours := 0.0;
       #ioRun_Time_S.Run_Time.Years := 0.0;
       #ioRun_Time_S.Run_Time.Seconds := 0;
       #ioRun_Time_S.Run_Time.Minutes := 0;
   END_IF;
END_REGION

REGION Network 3: Set Time
   RUNG wire#powerrail
      Contact( #tVKE1 )
      Contact( #iSetTime )
      wire#w1
      { S7_GenerateENO := "TRUE" } Move(in := #ioRun_Time_C.run_Time.seconds, out1 => #ioRun_Time_S.Run_Time.Seconds)
   END_RUNG
   RUNG wire#w1
      { S7_GenerateENO := "TRUE" } Move(in := #ioRun_Time_C.run_Time.minutes, out1 => #ioRun_Time_S.Run_Time.Minutes)
   END_RUNG
   RUNG wire#w1
      { S7_GenerateENO := "TRUE" } Move(in := #ioRun_Time_C.run_Time.hours, out1 => #ioRun_Time_S.Run_Time.Hours)
   END_RUNG
   RUNG wire#w1
      { S7_GenerateENO := "TRUE" } Move(in := #ioRun_Time_C.run_Time.days, out1 => #ioRun_Time_S.Run_Time.Days)
   END_RUNG
   RUNG wire#w1
      { S7_GenerateENO := "TRUE" } Move(in := #ioRun_Time_C.run_Time.years, out1 => #ioRun_Time_S.Run_Time.Years)
   END_RUNG
   // the same network as SCL:
   IF #tVKE1 AND #iSetTime THEN
       #ioRun_Time_S.Run_Time.Seconds := #ioRun_Time_C.run_Time.seconds;
       #ioRun_Time_S.Run_Time.Minutes := #ioRun_Time_C.run_Time.minutes;
       #ioRun_Time_S.Run_Time.Hours := #ioRun_Time_C.run_Time.hours;
       #ioRun_Time_S.Run_Time.Days := #ioRun_Time_C.run_Time.days;
       #ioRun_Time_S.Run_Time.Years := #ioRun_Time_C.run_Time.years;
   END_IF;
END_REGION

REGION Network 4: Check if Motor is running
   RUNG wire#powerrail
      Contact( #"iMotor Run Freedback" )
      Coil( #sMotoris_Enabled )
   END_RUNG
   // the same network as SCL:
   #sMotoris_Enabled := #"iMotor Run Freedback";
END_REGION

REGION Network 5: Start counting as long as Motor running
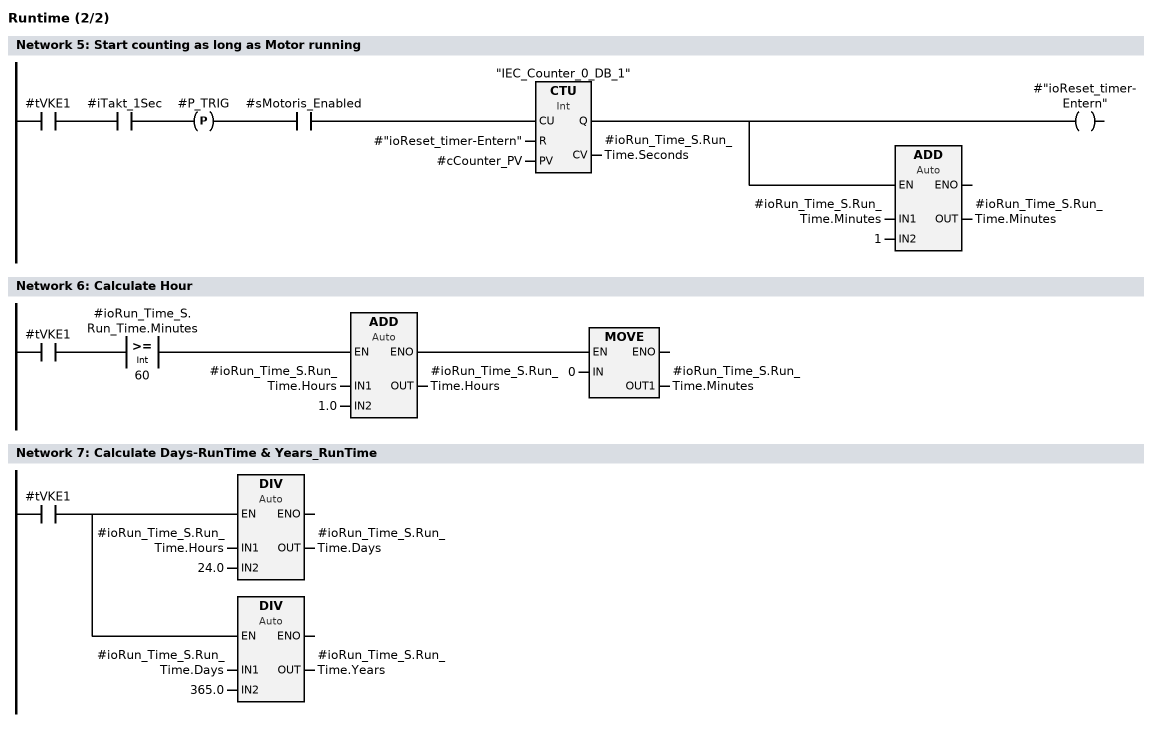
   RUNG wire#powerrail
      Contact( #tVKE1 )
      Contact( #iTakt_1Sec )
      P_Trig( #P_TRIG )
      Contact( #sMotoris_Enabled )
      { S7_Templates := "value_type := Int" } "IEC_Counter_0_DB_1".CTU(r := #"ioReset_timer-Entern", pv := #cCounter_PV, cv => #ioRun_Time_S.Run_Time.Seconds)
      wire#w1
      Coil( #"ioReset_timer-Entern" )
   END_RUNG
   RUNG wire#w1
      { S7_GenerateENO := "TRUE" } Add(in1 := #ioRun_Time_S.Run_Time.Minutes, in2 := 1, out => #ioRun_Time_S.Run_Time.Minutes)
   END_RUNG
   // the same network as SCL:
   #_w1 := #tVKE1 AND #iTakt_1Sec;
   #_w2 := #_w1 AND NOT #P_TRIG;   // rising edge
   #P_TRIG := #_w1;
   "IEC_Counter_0_DB_1".CTU(CU := #_w2 AND #sMotoris_Enabled,
                           R := #"ioReset_timer-Entern",
                           PV := #cCounter_PV,
                           CV => #ioRun_Time_S.Run_Time.Seconds);
   #"ioReset_timer-Entern" := "IEC_Counter_0_DB_1".Q;
   IF "IEC_Counter_0_DB_1".Q THEN
       #ioRun_Time_S.Run_Time.Minutes := #ioRun_Time_S.Run_Time.Minutes + 1;
   END_IF;
END_REGION

REGION Network 6: Calculate Hour
   RUNG wire#powerrail
      Contact( #tVKE1 )
      { S7_Templates := "SrcType := Int" } GE_Contact(in1 := #ioRun_Time_S.Run_Time.Minutes, in2 := 60)
      { S7_GenerateENO := "TRUE" } Add(in1 := #ioRun_Time_S.Run_Time.Hours, in2 := 1.0, out => #ioRun_Time_S.Run_Time.Hours)
      { S7_GenerateENO := "TRUE" } Move(in := 0, out1 => #ioRun_Time_S.Run_Time.Minutes)
   END_RUNG
   // the same network as SCL:
   // ENO of a box is taken as its EN; it also drops when the box reports an error
   IF #tVKE1 AND (#ioRun_Time_S.Run_Time.Minutes >= 60) THEN
       #ioRun_Time_S.Run_Time.Hours := #ioRun_Time_S.Run_Time.Hours + 1.0;
       #ioRun_Time_S.Run_Time.Minutes := 0;
   END_IF;
END_REGION

REGION Network 7: Calculate Days-RunTime & Years_RunTime
   RUNG wire#powerrail
      Contact( #tVKE1 )
      wire#w1
      { S7_GenerateENO := "TRUE" } Div(in1 := #ioRun_Time_S.Run_Time.Hours, in2 := 24.0, out => #ioRun_Time_S.Run_Time.Days)
   END_RUNG
   RUNG wire#w1
      { S7_GenerateENO := "TRUE" } Div(in1 := #ioRun_Time_S.Run_Time.Days, in2 := 365.0, out => #ioRun_Time_S.Run_Time.Years)
   END_RUNG
   // the same network as SCL:
   IF #tVKE1 THEN
       #ioRun_Time_S.Run_Time.Days := #ioRun_Time_S.Run_Time.Hours / 24.0;
       #ioRun_Time_S.Run_Time.Years := #ioRun_Time_S.Run_Time.Days / 365.0;
   END_IF;
END_REGION

REGION Network 8: End
END_REGION
END_FUNCTION_BLOCK

FUNCTION_BLOCK "timer ON"   // FB6, LAD
{ S7_Optimized_Access := 'TRUE' }
// stored: SetENOAutomatically false
   VAR_OUTPUT
      second : Int;
      minutes : Int;
      hours : Real;
      days : Real;
      years : Real;
   END_VAR
   VAR
      P_TRIG : Bool;
      Timer_R : Bool;
   END_VAR
   VAR_TEMP
      tVKE1 : Bool;
      tVKE0 : Bool;
   END_VAR
   VAR_TEMP   // added for the SCL form of the ladder/FBD networks
      _w1 : Bool;
   END_VAR
BEGIN

REGION Network 1: Create tVKE1 Netzwek
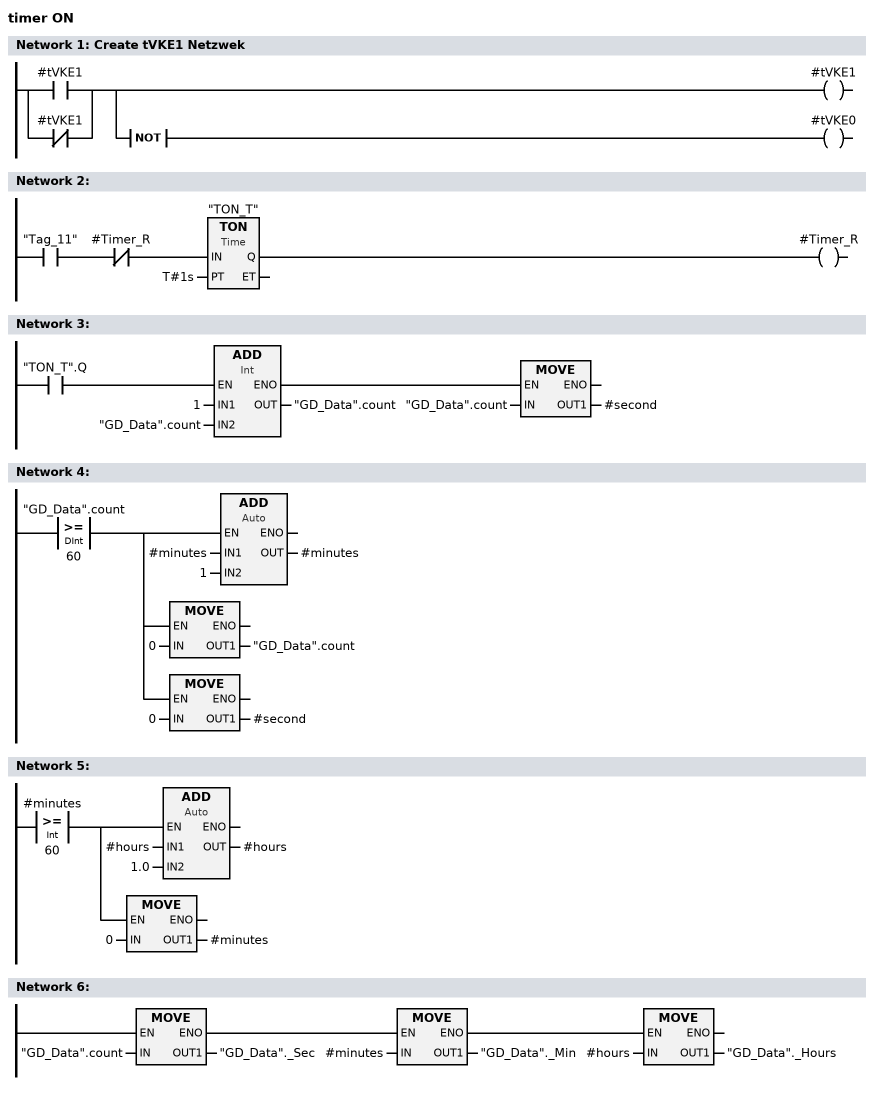
   RUNG wire#powerrail
      Contact( #tVKE1 )
      wire#w1
      Coil( #tVKE1 )
   END_RUNG
   RUNG wire#powerrail
      I_Contact( #tVKE1 )
   END_RUNG wire#w1
   RUNG wire#w1
      Not()
      Coil( #tVKE0 )
   END_RUNG
   // the same network as SCL:
   #tVKE1 := #tVKE1 OR NOT #tVKE1;
   #tVKE0 := NOT #tVKE1;
END_REGION

REGION Network 2
   RUNG wire#powerrail
      Contact( "Tag_11" )
      I_Contact( #Timer_R )
      { S7_Templates := "time_type := Time" } "TON_T".TON(pt := T#1s, et =>)
      Coil( #Timer_R )
   END_RUNG
   // the same network as SCL:
   "TON_T".TON(PT := T#1s, IN := "Tag_11" AND NOT #Timer_R);
   #Timer_R := "TON_T".Q;
END_REGION

REGION Network 3
   RUNG wire#powerrail
      Contact( "TON_T".Q )
      { S7_Templates := "SrcType := Int"; S7_GenerateENO := "TRUE" } Add(in1 := 1, in2 := "GD_Data".count, out => "GD_Data".count)
      { S7_GenerateENO := "TRUE" } Move(in := "GD_Data".count, out1 => #second)
   END_RUNG
   // the same network as SCL:
   // ENO of a box is taken as its EN; it also drops when the box reports an error
   IF "TON_T".Q THEN
       "GD_Data".count := 1 + "GD_Data".count;
       #second := "GD_Data".count;
   END_IF;
END_REGION

REGION Network 4
   RUNG wire#powerrail
      { S7_Templates := "SrcType := DInt" } GE_Contact(in1 := "GD_Data".count, in2 := 60)
      wire#w1
      { S7_GenerateENO := "TRUE" } Add(in1 := #minutes, in2 := 1, out => #minutes)
   END_RUNG
   RUNG wire#w1
      { S7_GenerateENO := "TRUE" } Move(in := 0, out1 => "GD_Data".count)
   END_RUNG
   RUNG wire#w1
      { S7_GenerateENO := "TRUE" } Move(in := 0, out1 => #second)
   END_RUNG
   // the same network as SCL:
   IF "GD_Data".count >= 60 THEN #minutes := #minutes + 1; END_IF;
   #_w1 := "GD_Data".count >= 60;
   IF #_w1 THEN
       "GD_Data".count := 0;
       #second := 0;
   END_IF;
END_REGION

REGION Network 5
   RUNG wire#powerrail
      { S7_Templates := "SrcType := Int" } GE_Contact(in1 := #minutes, in2 := 60)
      wire#w1
      { S7_GenerateENO := "TRUE" } Add(in1 := #hours, in2 := 1.0, out => #hours)
   END_RUNG
   RUNG wire#w1
      { S7_GenerateENO := "TRUE" } Move(in := 0, out1 => #minutes)
   END_RUNG
   // the same network as SCL:
   IF #minutes >= 60 THEN
       #hours := #hours + 1.0;
       #minutes := 0;
   END_IF;
END_REGION

REGION Network 6
   RUNG wire#powerrail
      { S7_GenerateENO := "TRUE" } Move(in := "GD_Data".count, out1 => "GD_Data"._Sec)
      { S7_GenerateENO := "TRUE" } Move(in := #minutes, out1 => "GD_Data"._Min)
      { S7_GenerateENO := "TRUE" } Move(in := #hours, out1 => "GD_Data"._Hours)
   END_RUNG
   // the same network as SCL:
   // ENO of a box is taken as its EN; it also drops when the box reports an error
   "GD_Data"._Sec := "GD_Data".count;
   "GD_Data"._Min := #minutes;
   "GD_Data"._Hours := #hours;
END_REGION
END_FUNCTION_BLOCK

FUNCTION "Bit_To_Word" : Void   // FC2, LAD
{ S7_Optimized_Access := 'TRUE' }
// stored: SetENOAutomatically false
   VAR_INPUT
      BIT : "UDT_Flowmeter_Stoe";
   END_VAR
   VAR_OUTPUT
      Out_I : Int;
   END_VAR
   VAR_TEMP
      Out_W : Word;
   END_VAR
BEGIN

REGION Network 1 (SCL)
   #Out_W :=0;

   IF #BIT."No Flow Detected" THEN
       #Out_W := #Out_W OR W#16#1;
   END_IF;

   IF #BIT."Flow Rate Too Low" THEN
       #Out_W := #Out_W OR W#16#2;
   END_IF;

   IF #BIT."Flow Rate Too Hight" THEN
       #Out_W := #Out_W OR W#16#4;
   END_IF;

   IF #BIT."Sensor CH1_wBreak" THEN
       #Out_W := #Out_W OR W#16#8;
   END_IF;

   IF #BIT."Sensor CH2_wBreak" THEN
       #Out_W := #Out_W OR W#16#10;
   END_IF;

   IF #BIT."Temprature Above Limit" THEN
       #Out_W := #Out_W OR W#16#20;
   END_IF;

   IF #BIT."Flow Out Of Range" THEN
       #Out_W := #Out_W OR W#16#40;
   END_IF;

   IF #BIT."Calibration Error" THEN
       #Out_W := #Out_W OR W#16#80;
   END_IF;

   IF   #BIT."Air Bubles Detected"    THEN
       #Out_W := #Out_W OR W#16#100;
   END_IF;

   IF #BIT."Temprature Out Of Range" THEN
       #Out_W := #Out_W OR W#16#200;
   END_IF;

   IF #BIT."Temprature Below Limit" THEN
       #Out_W := #Out_W OR W#16#400;
   END_IF;

   IF #BIT."Reverse Flow Detected" THEN
       #Out_W := #Out_W OR W#16#800;
   END_IF;

   IF #BIT."Communcation Error" THEN
       #Out_W := #Out_W OR W#16#1000;
   END_IF;

   IF #BIT."Clogging or Blockage" THEN
       #Out_W := #Out_W OR W#16#2000;
   END_IF;

   IF #BIT."Sensor Overheating" THEN
       #Out_W := #Out_W OR W#16#4000;
   END_IF;

   IF #BIT."Dirty Sensor" THEN
       #Out_W := #Out_W OR W#16#8000;
   END_IF;

   #Out_I := WORD_TO_INT(#Out_W);
END_REGION
END_FUNCTION

FUNCTION "Startup_FC" : Void   // FC1, LAD
{ S7_Optimized_Access := 'TRUE' }
// stored: SetENOAutomatically false
   VAR_TEMP
      ResetCount_0 : DInt;
      ResetCount_1 : DInt;
      P_Trig : Bool;
   END_VAR
   VAR_TEMP   // added for the SCL form of the ladder/FBD networks
      _w1 : Bool;
   END_VAR
BEGIN

REGION Network 1
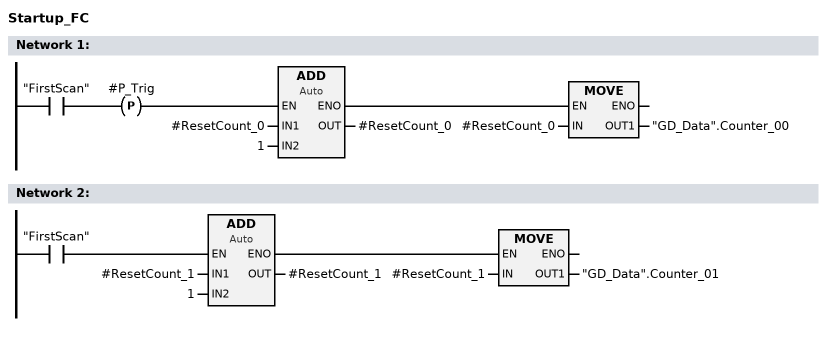
   RUNG wire#powerrail
      Contact( "FirstScan" )
      P_Trig( #P_Trig )
      { S7_GenerateENO := "TRUE" } Add(in1 := #ResetCount_0, in2 := 1, out => #ResetCount_0)
      { S7_GenerateENO := "TRUE" } Move(in := #ResetCount_0, out1 => "GD_Data".Counter_00)
   END_RUNG
   // the same network as SCL:
   // ENO of a box is taken as its EN; it also drops when the box reports an error
   #_w1 := "FirstScan" AND NOT #P_Trig;   // rising edge
   #P_Trig := "FirstScan";
   IF #_w1 THEN
       #ResetCount_0 := #ResetCount_0 + 1;
       "GD_Data".Counter_00 := #ResetCount_0;
   END_IF;
END_REGION

REGION Network 2
   RUNG wire#powerrail
      Contact( "FirstScan" )
      { S7_GenerateENO := "TRUE" } Add(in1 := #ResetCount_1, in2 := 1, out => #ResetCount_1)
      { S7_GenerateENO := "TRUE" } Move(in := #ResetCount_1, out1 => "GD_Data".Counter_01)
   END_RUNG
   // the same network as SCL:
   // ENO of a box is taken as its EN; it also drops when the box reports an error
   IF "FirstScan" THEN
       #ResetCount_1 := #ResetCount_1 + 1;
       "GD_Data".Counter_01 := #ResetCount_1;
   END_IF;
END_REGION
END_FUNCTION

FUNCTION_BLOCK "Block_1"
{ S7_Optimized_Access := 'TRUE' }
VERSION : 0.1
   VAR_INPUT 
      MotorRun : Bool;
      OneHzPulse : Bool;
      ResetTotals : Bool;
   END_VAR

   VAR_OUTPUT 
      Seconds : UDInt;
      Minutes : UDInt;
      Hours : UDInt;
      TotalSeconds : UDInt;
      TotalHours : UDInt;
   END_VAR

   VAR_TEMP 
      pulsePrev : Bool;
   END_VAR


BEGIN
	
	
	IF #ResetTotals THEN
	    #Seconds := 0;
	    #Minutes := 0;
	    #Hours := 0;
	    #TotalSeconds := 0;
	END_IF;
	
	
	IF #OneHzPulse AND  #pulsePrev THEN
	    IF #MotorRun THEN
	        "IEC_Counter_0_DB".CTU(CU:=#OneHzPulse,
	                               PV:=60);
	        
	       
	        #Seconds := #Seconds + 1;
	        #TotalSeconds := #TotalSeconds + 1;
	        
	        IF #Seconds >= 60 THEN
	            #Seconds := 0;
	            #Minutes := #Minutes + 1;
	        END_IF;
	        
	        IF #Minutes >= 60 THEN
	            #Minutes := 0;
	            #Hours := #Hours + 1;
	        END_IF;
	    END_IF;
	END_IF;
	
	
	#pulsePrev := #OneHzPulse;
	
	#TotalHours := UDINT_TO_REAL(#TotalSeconds) / 3600.0;
END_FUNCTION_BLOCK

DATA_BLOCK "FB_FlowMeter_DB_2"   // DB4
// stored: InstanceOfName FB_FlowMeter_FDH32, InstanceOfType FB
"FB_FlowMeter_FDH32"
BEGIN
END_DATA_BLOCK

DATA_BLOCK "FB_Fuel_Stand_DB"   // DB8
// stored: InstanceOfName FB_Fuel_Stand, InstanceOfType FB
"FB_Fuel_Stand"
BEGIN
END_DATA_BLOCK

DATA_BLOCK "Runtime_DB"   // DB7
// stored: InstanceOfName Runtime, InstanceOfType FB
"Runtime"
BEGIN
END_DATA_BLOCK

DATA_BLOCK "Startup_FB_DB"   // DB14
// stored: InstanceOfName Startup_FB, InstanceOfType FB
"Startup_FB"
BEGIN
END_DATA_BLOCK

DATA_BLOCK "timer ON_DB"   // DB9
// stored: InstanceOfName timer ON, InstanceOfType FB
"timer ON"
BEGIN
END_DATA_BLOCK

DATA_BLOCK "IEC_Counter_0_DB"   // DB5
{ S7_Optimized_Access := 'TRUE' }
// stored: InstanceOfName IEC_COUNTER, OfSystemLibElement IEC_COUNTER, OfSystemLibVersion 1.0
"IEC_COUNTER"
   // VAR RETAIN
   //    CU : Bool;
   //    CD : Bool;
   //    R : Bool;
   //    LD : Bool;
   //    QU : Bool;
   //    QD : Bool;
   //    PV : Int;
   //    CV : Int;
   // END_VAR
BEGIN
END_DATA_BLOCK

DATA_BLOCK "IEC_Counter_0_DB_1"   // DB6
{ S7_Optimized_Access := 'TRUE' }
// stored: InstanceOfName IEC_COUNTER, OfSystemLibElement IEC_COUNTER, OfSystemLibVersion 1.0
"IEC_COUNTER"
   // VAR RETAIN
   //    CU : Bool;
   //    CD : Bool;
   //    R : Bool;
   //    LD : Bool;
   //    QU : Bool;
   //    QD : Bool;
   //    PV : Int;
   //    CV : Int;
   // END_VAR
BEGIN
END_DATA_BLOCK

DATA_BLOCK "R_TRIG_DB"   // DB13
// stored: InstanceOfName R_TRIG, OfSystemLibElement R_TRIG, OfSystemLibVersion 1.0
"R_TRIG"
   // VAR_INPUT
   //    CLK : Bool;
   // END_VAR
   // VAR_OUTPUT
   //    Q : Bool;
   // END_VAR
   // VAR
   //    Stat_Bit : Bool;
   // END_VAR
BEGIN
END_DATA_BLOCK

DATA_BLOCK "TON_T"   // DB10
{ S7_Optimized_Access := 'TRUE' }
// stored: InstanceOfName IEC_TIMER, OfSystemLibElement IEC_TIMER, OfSystemLibVersion 1.0
"IEC_TIMER"
   // VAR
   //    PT : Time;
   //    ET { ExternalWritable := 'False'} : Time;
   //    IN : Bool;
   //    Q { ExternalWritable := 'False'} : Bool;
   // END_VAR
BEGIN
END_DATA_BLOCK
